KUKA KRL program: MyProgram_190().src

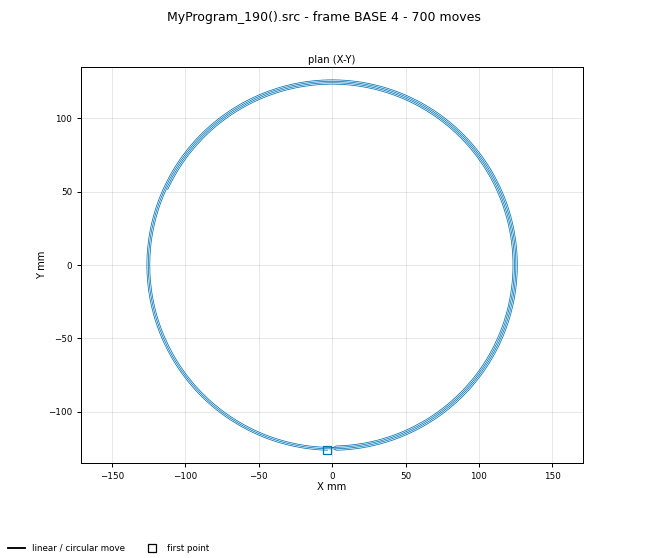
[picture p0: tool path of MyProgram_190().src in frame BASE 4, 700 of 700 moves have a stored position in this frame; points joined in program order, loops and branches not executed]
&ACCESS RVP
&REL 1
&PARAM TEMPLATE = C:\KRC\Roboter\Template\vorgabe
&PARAM EDITMASK = *
DEF MyProgram_190()
; ---- Setting reference (Base) ----
$BASE = BASE_DATA[4]

; --------------------------
; ---- Setting tool (TCP) ----
$TOOL = TOOL_DATA[3]
; --------------------------

$VEL.CP = VEL_APROX_PRINT
Startdeposition()
$VEL.CP = VEL_PRINT
LIN {X -3.1843,Y -126.111,Z 138,A -95.0934,B 24.9653,C -1.3617,E1 24.9951,E2 181.5075} C_DIS
LIN {X -7.0437,Y -125.9559,Z 138,A -96.9383,B 24.9655,C -1.3571,E1 24.9899,E2 183.3636} C_DIS
LIN {X -10.906,Y -125.6787,Z 138,A -98.6571,B 24.9654,C -1.3591,E1 24.9851,E2 185.0783} C_DIS
LIN {X -14.9041,Y -125.2671,Z 138,A -100.425,B 24.9652,C -1.3622,E1 24.9803,E2 186.8401} C_DIS
LIN {X -18.9665,Y -124.7171,Z 138,A -102.292,B 24.9652,C -1.3624,E1 24.9751,E2 188.7082} C_DIS
LIN {X -22.3988,Y -124.1462,Z 138,A -103.9323,B 24.9654,C -1.36,E1 24.9706,E2 190.3557} C_DIS
LIN {X -26.4694,Y -123.3424,Z 138,A -105.7239,B 24.9651,C -1.3653,E1 24.9657,E2 192.1369} C_DIS
LIN {X -29.6887,Y -122.6073,Z 138,A -107.3057,B 24.9652,C -1.3622,E1 24.9614,E2 193.7283} C_DIS
LIN {X -33.587,Y -121.5977,Z 138,A -108.947,B 24.9647,C -1.3723,E1 24.957,E2 195.3479} C_DIS
LIN {X -36.4143,Y -120.7816,Z 138,A -110.4707,B 24.9651,C -1.3643,E1 24.9529,E2 196.8933} C_DIS
LIN {X -39.9945,Y -119.6427,Z 138,A -112.121,B 24.9649,C -1.3683,E1 24.9485,E2 198.537} C_DIS
LIN {X -43.772,Y -118.3139,Z 138,A -113.9865,B 24.9649,C -1.3677,E1 24.9436,E2 200.4077} C_DIS
LIN {X -47.2767,Y -116.9565,Z 138,A -115.674,B 24.9649,C -1.3703,E1 24.9392,E2 202.0925} C_DIS
LIN {X -51.142,Y -115.3193,Z 138,A -117.5849,B 24.9647,C -1.3722,E1 24.9343,E2 204.0035} C_DIS
LIN {X -54.3155,Y -113.8583,Z 138,A -119.1216,B 24.9645,C -1.3765,E1 24.9304,E2 205.534} C_DIS
LIN {X -56.9474,Y -112.5654,Z 138,A -120.5382,B 24.9646,C -1.3741,E1 24.9269,E2 206.9598} C_DIS
LIN {X -61.2751,Y -110.2712,Z 138,A -122.6888,B 24.9643,C -1.3806,E1 24.9216,E2 209.1011} C_DIS
LIN {X -69.1084,Y -105.539,Z 138,A -127.0017,B 24.9643,C -1.3796,E1 24.9113,E2 213.4299} C_DIS
LIN {X -72.9275,Y -102.9369,Z 138,A -129.0758,B 24.9641,C -1.3843,E1 24.9066,E2 215.5} C_DIS
LIN {X -76.0268,Y -100.6691,Z 138,A -130.7644,B 24.9638,C -1.39,E1 24.9028,E2 217.181} C_DIS
LIN {X -78.4458,Y -98.7959,Z 138,A -132.3156,B 24.9641,C -1.385,E1 24.8994,E2 218.7496} C_DIS
LIN {X -82.0474,Y -95.8265,Z 138,A -134.3821,B 24.9637,C -1.3916,E1 24.8949,E2 220.8085} C_DIS
LIN {X -85.3051,Y -92.9376,Z 138,A -136.3149,B 24.9634,C -1.3977,E1 24.891,E2 222.7345} C_DIS
LIN {X -88.4698,Y -89.9305,Z 138,A -138.3203,B 24.9632,C -1.4009,E1 24.8869,E2 224.7408} C_DIS
LIN {X -91.4952,Y -86.8512,Z 138,A -140.3496,B 24.9632,C -1.402,E1 24.883,E2 226.776} C_DIS
LIN {X -94.065,Y -84.0604,Z 138,A -142.0826,B 24.963,C -1.4055,E1 24.8797,E2 228.5084} C_DIS
LIN {X -96.9286,Y -80.7424,Z 138,A -144.0584,B 24.9627,C -1.4109,E1 24.8762,E2 230.4805} C_DIS
LIN {X -99.5575,Y -77.4772,Z 138,A -145.9489,B 24.9624,C -1.4161,E1 24.8729,E2 232.3674} C_DIS
LIN {X -102.1418,Y -74.0365,Z 138,A -147.8756,B 24.9621,C -1.4223,E1 24.8697,E2 234.2887} C_DIS
LIN {X -104.5441,Y -70.6039,Z 138,A -149.8202,B 24.9619,C -1.4253,E1 24.8666,E2 236.2358} C_DIS
LIN {X -106.2939,Y -67.941,Z 138,A -151.3596,B 24.9619,C -1.4249,E1 24.8643,E2 237.7838} C_DIS
LIN {X -108.6351,Y -64.1314,Z 138,A -153.3025,B 24.9615,C -1.4344,E1 24.8615,E2 239.7142} C_DIS
LIN {X -110.5296,Y -60.8086,Z 138,A -155.0863,B 24.9613,C -1.4371,E1 24.8591,E2 241.5009} C_DIS
LIN {X -112.4396,Y -57.1946,Z 138,A -156.6495,B 24.9603,C -1.4556,E1 24.8571,E2 243.0282} C_DIS
LIN {X -114.1727,Y -53.6571,Z 138,A -158.7538,B 24.9608,C -1.4464,E1 24.8545,E2 245.1659} C_DIS
LIN {X -115.613,Y -50.4751,Z 138,A -160.2363,B 24.9603,C -1.4558,E1 24.8528,E2 246.6343} C_DIS
LIN {X -116.8237,Y -47.6062,Z 138,A -161.6588,B 24.9601,C -1.4595,E1 24.8513,E2 248.0557} C_DIS
LIN {X -118.3738,Y -43.612,Z 138,A -163.7518,B 24.9601,C -1.4587,E1 24.8492,E2 250.1624} C_DIS
LIN {X -119.6109,Y -40.0901,Z 138,A -165.3569,B 24.9596,C -1.468,E1 24.8478,E2 251.7547} C_DIS
LIN {X -120.5433,Y -37.193,Z 138,A -166.7446,B 24.9594,C -1.4719,E1 24.8466,E2 253.1408} C_DIS
LIN {X -121.4782,Y -34.0144,Z 138,A -168.2107,B 24.9591,C -1.4783,E1 24.8455,E2 254.6002} C_DIS
LIN {X -122.4907,Y -30.1723,Z 138,A -170.1494,B 24.9591,C -1.4779,E1 24.8441,E2 256.5511} C_DIS
LIN {X -123.8233,Y -24.1234,Z 138,A -172.9553,B 24.9586,C -1.4872,E1 24.8425,E2 259.3516} C_DIS
LIN {X -124.6687,Y -19.2791,Z 138,A -175.1858,B 24.9582,C -1.4945,E1 24.8415,E2 261.5779} C_DIS
LIN {X -125.1856,Y -15.5875,Z 138,A -176.8705,B 24.9578,C -1.5003,E1 24.8409,E2 263.2589} C_DIS
LIN {X -125.5705,Y -12.0845,Z 138,A -178.3017,B 24.9571,C -1.5131,E1 24.8405,E2 264.6681} C_DIS
LIN {X -125.7984,Y -9.4238,Z 138,A -179.776,B 24.9575,C -1.5053,E1 24.8401,E2 266.1698} C_DIS
LIN {X -126.0383,Y -5.3412,Z 138,A 178.3913,B 24.9571,C -1.5125,E1 24.8399,E2 267.9965} C_DIS
LIN {X -126.1439,Y -1.4652,Z 138,A 176.6709,B 24.9567,C -1.5201,E1 24.8398,E2 269.7091} C_DIS
LIN {X -126.1274,Y 2.4575,Z 138,A 174.9144,B 24.9563,C -1.527,E1 24.8398,E2 271.4596} C_DIS
LIN {X -125.9954,Y 6.2594,Z 138,A 173.1294,B 24.9561,C -1.5302,E1 24.84,E2 273.2478} C_DIS
LIN {X -125.7286,Y 10.3157,Z 138,A 171.4908,B 24.9552,C -1.5455,E1 24.8404,E2 274.8597} C_DIS
LIN {X -125.3625,Y 14.0922,Z 138,A 169.4724,B 24.9557,C -1.538,E1 24.8409,E2 276.9082} C_DIS
LIN {X -125.0413,Y 16.6956,Z 138,A 168.198,B 24.9557,C -1.5382,E1 24.8414,E2 278.1897} C_DIS
LIN {X -124.3839,Y 21.0404,Z 138,A 166.2733,B 24.9551,C -1.5479,E1 24.8423,E2 280.1028} C_DIS
LIN {X -123.728,Y 24.6098,Z 138,A 164.6559,B 24.9547,C -1.5546,E1 24.8431,E2 281.7136} C_DIS
LIN {X -123.0002,Y 28.0159,Z 138,A 162.8239,B 24.9551,C -1.5486,E1 24.8442,E2 283.5706} C_DIS
LIN {X -121.846,Y 32.6729,Z 138,A 160.8635,B 24.9541,C -1.5654,E1 24.8456,E2 285.5025} C_DIS
LIN {X -120.7193,Y 36.6178,Z 138,A 159.0027,B 24.9537,C -1.5715,E1 24.847,E2 287.3595} C_DIS
LIN {X -119.6782,Y 39.8879,Z 138,A 157.4553,B 24.9534,C -1.577,E1 24.8484,E2 288.9027} C_DIS
LIN {X -118.4195,Y 43.489,Z 138,A 155.6809,B 24.9532,C -1.5805,E1 24.85,E2 290.6787} C_DIS
LIN {X -117.115,Y 46.8834,Z 138,A 153.9246,B 24.9532,C -1.5811,E1 24.8518,E2 292.4437} C_DIS
LIN {X -115.3426,Y 51.0899,Z 138,A 152.1114,B 24.9521,C -1.5991,E1 24.8538,E2 294.2238} C_DIS
LIN {X -112.9708,Y 56.1391,Z 138,A 148.6942,B 24.954,C -1.5675,E1 24.8581,E2 297.735} C_DIS
LIN {X -110.5428,Y 60.7845,Z 138,A 146.6018,B 24.9528,C -1.5873,E1 24.8608,E2 299.7912} C_DIS
LIN {X -108.7408,Y 63.9515,Z 138,A 145.1814,B 24.9519,C -1.6026,E1 24.8628,E2 301.1824} C_DIS
LIN {X -106.4029,Y 67.7707,Z 138,A 143.1806,B 24.9514,C -1.61,E1 24.8657,E2 303.1759} C_DIS
LIN {X -103.8973,Y 71.5524,Z 138,A 141.1937,B 24.9509,C -1.6191,E1 24.8688,E2 305.1509} C_DIS
LIN {X -101.4707,Y 74.9543,Z 138,A 139.208,B 24.9508,C -1.6204,E1 24.8721,E2 307.1432} C_DIS
LIN {X -98.8671,Y 78.3563,Z 138,A 137.2836,B 24.9504,C -1.6267,E1 24.8754,E2 309.0618} C_DIS
LIN {X -96.2209,Y 81.5838,Z 138,A 135.3622,B 24.9502,C -1.6305,E1 24.8788,E2 310.9828} C_DIS
LIN {X -93.2585,Y 84.9545,Z 138,A 133.2981,B 24.9499,C -1.6346,E1 24.8826,E2 313.0465} C_DIS
LIN {X -90.3023,Y 88.0906,Z 138,A 131.3418,B 24.9496,C -1.6396,E1 24.8864,E2 314.9995} C_DIS
LIN {X -87.41,Y 90.9613,Z 138,A 129.4413,B 24.9495,C -1.6418,E1 24.8902,E2 316.9025} C_DIS
LIN {X -84.0588,Y 94.0664,Z 138,A 127.413,B 24.9491,C -1.6488,E1 24.8944,E2 318.9223} C_DIS
LIN {X -80.7619,Y 96.9125,Z 138,A 125.3839,B 24.9489,C -1.651,E1 24.8987,E2 320.9541} C_DIS
LIN {X -77.3811,Y 99.632,Z 138,A 123.4278,B 24.9486,C -1.656,E1 24.903,E2 322.9055} C_DIS
LIN {X -73.7304,Y 102.3636,Z 138,A 121.3155,B 24.9485,C -1.6585,E1 24.9077,E2 325.0194} C_DIS
LIN {X -70.0481,Y 104.9172,Z 138,A 119.304,B 24.9481,C -1.6636,E1 24.9124,E2 327.0253} C_DIS
LIN {X -66.2835,Y 107.3359,Z 138,A 117.2265,B 24.9481,C -1.6655,E1 24.9173,E2 329.1051} C_DIS
LIN {X -63.0471,Y 109.2678,Z 138,A 115.3202,B 24.9484,C -1.6597,E1 24.9219,E2 331.0309} C_DIS
LIN {X -60.2193,Y 110.8514,Z 138,A 114.0863,B 24.9475,C -1.6732,E1 24.9249,E2 332.2363} C_DIS
LIN {X -57.1335,Y 112.4707,Z 138,A 112.6236,B 24.947,C -1.6814,E1 24.9285,E2 333.6833} C_DIS
LIN {X -54.1653,Y 113.9301,Z 138,A 111.0462,B 24.947,C -1.6803,E1 24.9324,E2 335.2673} C_DIS
LIN {X -49.3542,Y 116.0976,Z 138,A 108.5307,B 24.9472,C -1.6784,E1 24.9389,E2 337.7935} C_DIS
LIN {X -45.9275,Y 117.4931,Z 138,A 106.9709,B 24.9467,C -1.6864,E1 24.9429,E2 339.3377} C_DIS
LIN {X -43.2268,Y 118.514,Z 138,A 105.6403,B 24.9467,C -1.6872,E1 24.9464,E2 340.669} C_DIS
LIN {X -37.0434,Y 120.5891,Z 138,A 102.7706,B 24.9462,C -1.6951,E1 24.954,E2 343.5252} C_DIS
LIN {X -34.1823,Y 121.4312,Z 138,A 101.3525,B 24.9462,C -1.6936,E1 24.9578,E2 344.9492} C_DIS
LIN {X -30.2186,Y 122.4795,Z 138,A 99.0393,B 24.9475,C -1.6744,E1 24.9642,E2 347.3115} C_DIS
LIN {X -26.6668,Y 123.2998,Z 138,A 97.5867,B 24.9468,C -1.6854,E1 24.9681,E2 348.7398} C_DIS
LIN {X -22.2034,Y 124.1812,Z 138,A 95.7017,B 24.9461,C -1.6955,E1 24.9732,E2 350.6026} C_DIS
LIN {X -18.2311,Y 124.8269,Z 138,A 93.8613,B 24.9461,C -1.6962,E1 24.9783,E2 352.4431} C_DIS
LIN {X -14.6843,Y 125.2933,Z 138,A 92.2052,B 24.9461,C -1.6957,E1 24.9829,E2 354.1015} C_DIS
LIN {X -10.7568,Y 125.6913,Z 138,A 90.446,B 24.946,C -1.6982,E1 24.9877,E2 355.8557} C_DIS
LIN {X -6.5893,Y 125.9788,Z 138,A 88.5503,B 24.946,C -1.699,E1 24.993,E2 357.7501} C_DIS
LIN {X -2.5849,Y 126.1252,Z 138,A 86.6906,B 24.946,C -1.6977,E1 24.9982,E2 359.6133} C_DIS
LIN {X 1.2278,Y 126.1459,Z 138,A 84.9358,B 24.946,C -1.6969,E1 25.0031,E2 361.3699} C_DIS
LIN {X 4.7952,Y 126.0596,Z 138,A 83.3843,B 24.9458,C -1.7004,E1 25.0074,E2 362.9127} C_DIS
LIN {X 8.6734,Y 125.8532,Z 138,A 81.5802,B 24.9459,C -1.6984,E1 25.0125,E2 364.7207} C_DIS
LIN {X 12.3307,Y 125.5469,Z 138,A 79.8631,B 24.9461,C -1.6958,E1 25.0173,E2 366.4429} C_DIS
LIN {X 16.3417,Y 125.0877,Z 138,A 78.1352,B 24.9458,C -1.7006,E1 25.022,E2 368.1583} C_DIS
LIN {X 20.3136,Y 124.5051,Z 138,A 76.2446,B 24.946,C -1.6967,E1 25.0273,E2 370.0561} C_DIS
LIN {X 23.9897,Y 123.8489,Z 138,A 74.5305,B 24.9461,C -1.6952,E1 25.032,E2 371.772} C_DIS
LIN {X 28.6252,Y 122.8611,Z 138,A 72.3822,B 24.9462,C -1.6943,E1 25.0378,E2 373.9197} C_DIS
LIN {X 32.2993,Y 121.9456,Z 138,A 70.8031,B 24.9458,C -1.7001,E1 25.0421,E2 375.4826} C_DIS
LIN {X 35.2724,Y 121.119,Z 138,A 69.395,B 24.9459,C -1.6987,E1 25.0458,E2 376.8914} C_DIS
LIN {X 38.3218,Y 120.1889,Z 138,A 67.8105,B 24.9464,C -1.6909,E1 25.0501,E2 378.4916} C_DIS
LIN {X 42.4475,Y 118.795,Z 138,A 65.9768,B 24.9461,C -1.6962,E1 25.0549,E2 380.3091} C_DIS
LIN {X 47.2661,Y 116.9608,Z 138,A 63.6076,B 24.9463,C -1.6925,E1 25.0611,E2 382.6818} C_DIS
LIN {X 50.697,Y 115.517,Z 138,A 61.8325,B 24.9467,C -1.6865,E1 25.0657,E2 384.4671} C_DIS
LIN {X 54.1241,Y 113.9497,Z 138,A 60.2039,B 24.9466,C -1.6885,E1 25.0698,E2 386.0866} C_DIS
LIN {X 59.137,Y 111.4316,Z 138,A 57.6397,B 24.9468,C -1.6843,E1 25.0761,E2 388.6537} C_DIS
LIN {X 61.5464,Y 110.1204,Z 138,A 55.6157,B 24.9493,C -1.6442,E1 25.0813,E2 390.7665} C_DIS
LIN {X 66.4381,Y 107.2399,Z 138,A 53.7538,B 24.9474,C -1.6755,E1 25.0855,E2 392.5486} C_DIS
LIN {X 70.3044,Y 104.7461,Z 138,A 51.6555,B 24.9476,C -1.6717,E1 25.0904,E2 394.6491} C_DIS
LIN {X 73.8549,Y 102.2734,Z 138,A 49.7166,B 24.9478,C -1.6696,E1 25.0948,E2 396.5862} C_DIS
LIN {X 77.3089,Y 99.6879,Z 138,A 47.8117,B 24.9478,C -1.6687,E1 25.0991,E2 398.4862} C_DIS
LIN {X 80.5283,Y 97.1059,Z 138,A 45.9147,B 24.9481,C -1.664,E1 25.1032,E2 400.3872} C_DIS
LIN {X 83.8428,Y 94.2597,Z 138,A 43.8929,B 24.9485,C -1.6581,E1 25.1074,E2 402.4149} C_DIS
LIN {X 86.381,Y 91.9388,Z 138,A 42.1429,B 24.9493,C -1.6454,E1 25.1111,E2 404.1877} C_DIS
LIN {X 88.7451,Y 89.6589,Z 138,A 40.8781,B 24.9488,C -1.6536,E1 25.1135,E2 405.4279} C_DIS
LIN {X 91.8682,Y 86.4558,Z 138,A 39.0098,B 24.9485,C -1.6573,E1 25.1171,E2 407.2793} C_DIS
LIN {X 94.718,Y 83.3243,Z 138,A 36.9318,B 24.9493,C -1.645,E1 25.121,E2 409.377} C_DIS
LIN {X 97.5231,Y 80.0228,Z 138,A 35.0003,B 24.9495,C -1.6421,E1 25.1245,E2 411.3065} C_DIS
LIN {X 100.1181,Y 76.7511,Z 138,A 33.2507,B 24.9493,C -1.6449,E1 25.1275,E2 413.0412} C_DIS
LIN {X 102.3611,Y 73.7339,Z 138,A 31.3767,B 24.9501,C -1.6321,E1 25.1306,E2 414.9364} C_DIS
LIN {X 104.915,Y 70.0514,Z 138,A 29.3991,B 24.9502,C -1.6298,E1 25.1337,E2 416.9097} C_DIS
LIN {X 107.3157,Y 66.3162,Z 138,A 27.3488,B 24.9507,C -1.6227,E1 25.1368,E2 418.9665} C_DIS
LIN {X 109.1543,Y 63.2431,Z 138,A 25.5345,B 24.9515,C -1.6087,E1 25.1394,E2 420.8045} C_DIS
LIN {X 110.7607,Y 60.3856,Z 138,A 24.3295,B 24.9509,C -1.619,E1 25.1409,E2 421.9788} C_DIS
LIN {X 114.4891,Y 52.973,Z 138,A 20.642,B 24.9513,C -1.6124,E1 25.1455,E2 425.6622} C_DIS
LIN {X 115.8897,Y 49.835,Z 138,A 19.048,B 24.9517,C -1.6061,E1 25.1473,E2 427.2622} C_DIS
LIN {X 117.448,Y 46.0433,Z 138,A 17.2365,B 24.9518,C -1.6032,E1 25.1492,E2 429.0707} C_DIS
LIN {X 118.7956,Y 42.4458,Z 138,A 15.2611,B 24.9529,C -1.5861,E1 25.1511,E2 431.0754} C_DIS
LIN {X 120.1635,Y 38.4011,Z 138,A 13.4636,B 24.9528,C -1.5874,E1 25.1526,E2 432.8595} C_DIS
LIN {X 121.6807,Y 33.2905,Z 138,A 11.0418,B 24.9532,C -1.5799,E1 25.1545,E2 435.2853} C_DIS
LIN {X 122.6042,Y 29.7014,Z 138,A 9.4799,B 24.9532,C -1.5809,E1 25.1556,E2 436.8358} C_DIS
LIN {X 123.5258,Y 25.6034,Z 138,A 7.5395,B 24.9536,C -1.5731,E1 25.1567,E2 438.7832} C_DIS
LIN {X 124.1856,Y 22.179,Z 138,A 6.0159,B 24.9537,C -1.5712,E1 25.1575,E2 440.3024} C_DIS
LIN {X 124.8109,Y 18.3432,Z 138,A 4.1928,B 24.9543,C -1.5625,E1 25.1583,E2 442.1353} C_DIS
LIN {X 125.3007,Y 14.6229,Z 138,A 2.492,B 24.9546,C -1.5572,E1 25.1589,E2 443.8386} C_DIS
LIN {X 125.7021,Y 10.6293,Z 138,A 0.7505,B 24.9546,C -1.5555,E1 25.1593,E2 445.5738} C_DIS
LIN {X 125.9762,Y 6.6414,Z 138,A -1.0667,B 24.955,C -1.5494,E1 25.1596,E2 447.3944} C_DIS
LIN {X 126.1201,Y 2.8566,Z 138,A -2.8293,B 24.9555,C -1.5416,E1 25.1598,E2 449.165} C_DIS
LIN {X 126.1503,Y -0.69,Z 138,A -4.4682,B 24.9559,C -1.5348,E1 25.1598,E2 450.8101} C_DIS
LIN {X 126.0556,Y -4.899,Z 138,A -6.2874,B 24.9559,C -1.5334,E1 25.1596,E2 452.6219} C_DIS
LIN {X 125.8258,Y -9.049,Z 138,A -8.1294,B 24.9562,C -1.5295,E1 25.1593,E2 454.462} C_DIS
LIN {X 125.4968,Y -12.8441,Z 138,A -9.9084,B 24.9566,C -1.5213,E1 25.1588,E2 456.2499} C_DIS
LIN {X 125.0537,Y -16.6009,Z 138,A -11.5281,B 24.9566,C -1.5208,E1 25.1583,E2 457.8613} C_DIS
LIN {X 124.4813,Y -20.4567,Z 138,A -13.2807,B 24.957,C -1.5159,E1 25.1575,E2 459.6152} C_DIS
LIN {X 123.8791,Y -23.8316,Z 138,A -14.866,B 24.9573,C -1.5093,E1 25.1567,E2 461.2066} C_DIS
LIN {X 123.2436,Y -26.9272,Z 138,A -16.5653,B 24.9584,C -1.4909,E1 25.1557,E2 462.9394} C_DIS
LIN {X 121.9819,Y -32.1631,Z 138,A -18.7377,B 24.958,C -1.4972,E1 25.1542,E2 465.0844} C_DIS
LIN {X 121.0599,Y -35.4744,Z 138,A -20.6849,B 24.9594,C -1.4722,E1 25.1527,E2 467.0795} C_DIS
LIN {X 119.8982,Y -39.2273,Z 138,A -21.9524,B 24.9582,C -1.4932,E1 25.1517,E2 468.2903} C_DIS
LIN {X 118.1968,Y -44.0845,Z 138,A -24.2966,B 24.9587,C -1.4854,E1 25.1495,E2 470.6396} C_DIS
LIN {X 117.0448,Y -47.0577,Z 138,A -25.8717,B 24.9593,C -1.4743,E1 25.1478,E2 472.2323} C_DIS
LIN {X 115.4048,Y -50.9508,Z 138,A -27.6176,B 24.9591,C -1.4773,E1 25.1459,E2 473.9616} C_DIS
LIN {X 114.032,Y -53.9519,Z 138,A -29.2873,B 24.9599,C -1.4638,E1 25.1439,E2 475.6539} C_DIS
LIN {X 112.424,Y -57.2252,Z 138,A -30.8725,B 24.9599,C -1.4624,E1 25.142,E2 477.2339} C_DIS
LIN {X 110.6036,Y -60.6736,Z 138,A -32.6818,B 24.9603,C -1.4551,E1 25.1395,E2 479.051} C_DIS
LIN {X 108.4198,Y -64.4944,Z 138,A -34.6472,B 24.9606,C -1.4509,E1 25.1368,E2 481.0161} C_DIS
LIN {X 106.0835,Y -68.2696,Z 138,A -36.6913,B 24.961,C -1.4436,E1 25.1337,E2 483.0671} C_DIS
LIN {X 103.7128,Y -71.8198,Z 138,A -38.6197,B 24.9612,C -1.4387,E1 25.1307,E2 484.9977} C_DIS
LIN {X 101.248,Y -75.2542,Z 138,A -41.247,B 24.9634,C -1.3971,E1 25.1262,E2 487.7104} C_DIS
LIN {X 97.6826,Y -79.8276,Z 138,A -42.915,B 24.9612,C -1.4394,E1 25.1235,E2 489.2707} C_DIS
LIN {X 93.6621,Y -84.5097,Z 138,A -45.9515,B 24.9622,C -1.42,E1 25.1178,E2 492.3394} C_DIS
LIN {X 90.972,Y -87.3988,Z 138,A -47.6004,B 24.9621,C -1.4228,E1 25.1147,E2 493.9745} C_DIS
LIN {X 88.0571,Y -90.335,Z 138,A -49.9829,B 24.9637,C -1.3924,E1 25.1098,E2 496.4186} C_DIS
LIN {X 85.0001,Y -93.2171,Z 138,A -51.4919,B 24.9629,C -1.4082,E1 25.1068,E2 497.8843} C_DIS
LIN {X 81.6866,Y -96.1335,Z 138,A -53.4312,B 24.9629,C -1.4069,E1 25.1027,E2 499.8191} C_DIS
LIN {X 79.4361,Y -98.0018,Z 138,A -55.2722,B 24.9644,C -1.3778,E1 25.0986,E2 501.7217} C_DIS
LIN {X 75.8471,Y -100.8048,Z 138,A -56.7504,B 24.9631,C -1.4033,E1 25.0955,E2 503.1345} C_DIS
LIN {X 73.2379,Y -102.716,Z 138,A -58.6682,B 24.9645,C -1.3774,E1 25.091,E2 505.1067} C_DIS
LIN {X 69.9914,Y -104.955,Z 138,A -60.4202,B 24.9645,C -1.3758,E1 25.0869,E2 506.8567} C_DIS
LIN {X 66.7977,Y -107.0161,Z 138,A -61.7787,B 24.9638,C -1.391,E1 25.0838,E2 508.1748} C_DIS
LIN {X 63.2431,Y -109.1543,Z 138,A -63.7237,B 24.9641,C -1.3844,E1 25.0791,E2 510.1295} C_DIS
LIN {X 59.2938,Y -111.3493,Z 138,A -65.803,B 24.9644,C -1.3794,E1 25.074,E2 512.2146} C_DIS
LIN {X 56.0006,Y -113.0392,Z 138,A -67.2995,B 24.964,C -1.3859,E1 25.0703,E2 513.6917} C_DIS
LIN {X 53.0828,Y -114.4383,Z 138,A -68.672,B 24.9639,C -1.3884,E1 25.0669,E2 515.0547} C_DIS
LIN {X 50.3542,Y -115.6652,Z 138,A -70.1541,B 24.9643,C -1.3801,E1 25.063,E2 516.5528} C_DIS
LIN {X 47.3312,Y -116.9345,Z 138,A -71.6241,B 24.9643,C -1.3789,E1 25.0593,E2 518.0223} C_DIS
LIN {X 41.9125,Y -118.9859,Z 138,A -74.2561,B 24.9646,C -1.3753,E1 25.0524,E2 520.6574} C_DIS
LIN {X 38.2727,Y -120.2045,Z 138,A -75.9935,B 24.9646,C -1.3734,E1 25.0477,E2 522.3958} C_DIS
LIN {X 32.7287,Y -121.8311,Z 138,A -78.6274,B 24.9648,C -1.37,E1 25.0407,E2 525.0334} C_DIS
LIN {X 28.7378,Y -122.8353,Z 138,A -80.5606,B 24.9651,C -1.3649,E1 25.0354,E2 526.9759} C_DIS
LIN {X 25.136,Y -123.6209,Z 138,A -82.2903,B 24.9653,C -1.3606,E1 25.0306,E2 528.7134} C_DIS
LIN {X 20.8141,Y -124.4216,Z 138,A -84.0653,B 24.9648,C -1.37,E1 25.0258,E2 530.4644} C_DIS
LIN {X 17.6706,Y -124.907,Z 138,A -85.5773,B 24.9651,C -1.3656,E1 25.0216,E2 531.9853} C_DIS
LIN {X 13.8266,Y -125.3911,Z 138,A -87.3421,B 24.9651,C -1.3643,E1 25.0167,E2 533.7519} C_DIS
LIN {X 10.3306,Y -125.7273,Z 138,A -89.0133,B 24.9654,C -1.3597,E1 25.0121,E2 535.433} C_DIS
LIN {X 6.5028,Y -125.9831,Z 138,A -90.6761,B 24.9652,C -1.3629,E1 25.0074,E2 537.0877} C_DIS
LIN {X 2.7912,Y -126.1218,Z 138,A -92.4593,B 24.9655,C -1.3576,E1 25.0024,E2 538.883} C_DIS
LIN {X 2.7912,Y -126.1218,Z 138,A -92.4593,B 24.9655,C -1.3576,E1 25.0024,E2 538.883} C_DIS
Enddeposition()
LIN {X 0.8852,Y -125.1643,Z 138,A -93.1588,B 24.9642,C -1.3828,E1 25.0007,E2 539.5227} C_DIS
Startdeposition()
$VEL.CP = VEL_PRINT
LIN {X 3.3988,Y -125.1228,Z 138,A -91.394,B 24.9626,C -1.4132,E1 25.0058,E2 537.6863} C_DIS
LIN {X 7.3779,Y -124.9516,Z 138,A -89.5453,B 24.9625,C -1.4152,E1 25.0109,E2 535.8334} C_DIS
LIN {X 11.1676,Y -124.6712,Z 138,A -87.7011,B 24.9622,C -1.4212,E1 25.0161,E2 533.9759} C_DIS
LIN {X 15.0926,Y -124.2558,Z 138,A -85.9375,B 24.9622,C -1.4202,E1 25.021,E2 532.2161} C_DIS
LIN {X 19.2045,Y -123.6867,Z 138,A -84.1263,B 24.9624,C -1.4171,E1 25.026,E2 530.4137} C_DIS
LIN {X 23.2174,Y -122.9969,Z 138,A -82.0486,B 24.9617,C -1.4293,E1 25.0317,E2 528.3095} C_DIS
LIN {X 27.4372,Y -122.1253,Z 138,A -80.4647,B 24.9627,C -1.4117,E1 25.036,E2 526.7693} C_DIS
LIN {X 30.6364,Y -121.3615,Z 138,A -78.8102,B 24.9622,C -1.4206,E1 25.0405,E2 525.096} C_DIS
LIN {X 38.0234,Y -119.2534,Z 138,A -75.3255,B 24.9621,C -1.423,E1 25.0498,E2 521.6117} C_DIS
LIN {X 44.3504,Y -117.0488,Z 138,A -72.261,B 24.9619,C -1.4269,E1 25.0579,E2 518.5443} C_DIS
LIN {X 48.0056,Y -115.597,Z 138,A -70.3888,B 24.9615,C -1.4331,E1 25.0628,E2 516.6616} C_DIS
LIN {X 51.5068,Y -114.0805,Z 138,A -68.7642,B 24.9617,C -1.4296,E1 25.0669,E2 515.0492} C_DIS
LIN {X 54.1038,Y -112.8713,Z 138,A -67.398,B 24.9614,C -1.4345,E1 25.0704,E2 513.6749} C_DIS
LIN {X 57.3557,Y -111.2558,Z 138,A -65.6064,B 24.9609,C -1.4439,E1 25.0749,E2 511.8661} C_DIS
LIN {X 63.1409,Y -108.0782,Z 138,A -62.6695,B 24.9609,C -1.4451,E1 25.082,E2 508.9352} C_DIS
LIN {X 66.5896,Y -105.9881,Z 138,A -60.8077,B 24.9606,C -1.4494,E1 25.0864,E2 507.069} C_DIS
LIN {X 69.6045,Y -104.0327,Z 138,A -58.7802,B 24.9594,C -1.4724,E1 25.0913,E2 504.994} C_DIS
LIN {X 72.9163,Y -101.739,Z 138,A -57.6001,B 24.961,C -1.4421,E1 25.0938,E2 503.8894} C_DIS
LIN {X 75.1,Y -100.1385,Z 138,A -56.0972,B 24.9602,C -1.4583,E1 25.0972,E2 502.3537} C_DIS
LIN {X 79.9228,Y -96.3325,Z 138,A -52.699,B 24.9581,C -1.4949,E1 25.1047,E2 498.882} C_DIS
LIN {X 83.7699,Y -93.0071,Z 138,A -51.1055,B 24.9599,C -1.4624,E1 25.1079,E2 497.3716} C_DIS
LIN {X 88.404,Y -88.6137,Z 138,A -48.3499,B 24.96,C -1.4608,E1 25.1134,E2 494.631} C_DIS
LIN {X 92.6399,Y -84.1751,Z 138,A -45.3753,B 24.9592,C -1.4765,E1 25.1192,E2 491.6324} C_DIS
LIN {X 96.577,Y -79.6275,Z 138,A -42.6928,B 24.959,C -1.4801,E1 25.124,E2 488.9537} C_DIS
LIN {X 100.1693,Y -75.059,Z 138,A -40.1585,B 24.959,C -1.4808,E1 25.1284,E2 486.4296} C_DIS
LIN {X 101.7027,Y -72.967,Z 138,A -38.7235,B 24.958,C -1.497,E1 25.1308,E2 484.9635} C_DIS
LIN {X 104.0523,Y -69.5752,Z 138,A -36.8343,B 24.9577,C -1.5024,E1 25.1337,E2 483.0708} C_DIS
LIN {X 106.3973,Y -65.9337,Z 138,A -34.8597,B 24.9574,C -1.5077,E1 25.1367,E2 481.0937} C_DIS
LIN {X 108.4615,Y -62.48,Z 138,A -33.0225,B 24.9571,C -1.5129,E1 25.1393,E2 479.2536} C_DIS
LIN {X 110.1462,Y -59.4599,Z 138,A -31.4785,B 24.957,C -1.5156,E1 25.1413,E2 477.7113} C_DIS
LIN {X 112.0758,Y -55.7342,Z 138,A -29.6105,B 24.9568,C -1.5187,E1 25.1437,E2 475.8459} C_DIS
LIN {X 113.6426,Y -52.4642,Z 138,A -27.9747,B 24.9566,C -1.5226,E1 25.1456,E2 474.2099} C_DIS
LIN {X 115.874,Y -47.3359,Z 138,A -25.5598,B 24.9566,C -1.5229,E1 25.1483,E2 471.8074} C_DIS
LIN {X 117.391,Y -43.4367,Z 138,A -23.4333,B 24.9556,C -1.54,E1 25.1504,E2 469.6524} C_DIS
LIN {X 118.9827,Y -38.8687,Z 138,A -20.8684,B 24.9541,C -1.5655,E1 25.1527,E2 467.042} C_DIS
LIN {X 120.1431,Y -35.1112,Z 138,A -19.5632,B 24.9553,C -1.5453,E1 25.1537,E2 465.7918} C_DIS
LIN {X 121.1599,Y -31.4309,Z 138,A -16.993,B 24.9524,C -1.5942,E1 25.1556,E2 463.1212} C_DIS
LIN {X 122.4816,Y -25.8039,Z 138,A -15.2459,B 24.9547,C -1.5555,E1 25.1566,E2 461.4755} C_DIS
LIN {X 123.069,Y -22.84,Z 138,A -13.7051,B 24.9539,C -1.5683,E1 25.1574,E2 459.9136} C_DIS
LIN {X 123.6896,Y -19.1858,Z 138,A -12.1303,B 24.9539,C -1.5675,E1 25.1581,E2 458.3499} C_DIS
LIN {X 124.2349,Y -15.2682,Z 138,A -10.2593,B 24.9534,C -1.5766,E1 25.1588,E2 456.4684} C_DIS
LIN {X 124.6082,Y -11.8335,Z 138,A -8.7572,B 24.9534,C -1.5777,E1 25.1592,E2 454.9727} C_DIS
LIN {X 124.9277,Y -7.7667,Z 138,A -6.9056,B 24.953,C -1.583,E1 25.1595,E2 453.1195} C_DIS
LIN {X 125.1138,Y -3.7217,Z 138,A -5.0474,B 24.9527,C -1.5893,E1 25.1597,E2 451.2574} C_DIS
LIN {X 125.1709,Y 0.3093,Z 138,A -3.1114,B 24.952,C -1.6001,E1 25.1597,E2 449.3075} C_DIS
LIN {X 125.0876,Y 4.5231,Z 138,A -1.285,B 24.952,C -1.6011,E1 25.1597,E2 447.4897} C_DIS
LIN {X 124.9014,Y 8.1939,Z 138,A 0.4591,B 24.9514,C -1.6098,E1 25.1593,E2 445.7354} C_DIS
LIN {X 124.5576,Y 12.3608,Z 138,A 2.3148,B 24.9512,C -1.613,E1 25.1589,E2 443.8832} C_DIS
LIN {X 124.0998,Y 16.3235,Z 138,A 4.0783,B 24.9511,C -1.6157,E1 25.1583,E2 442.1238} C_DIS
LIN {X 123.5001,Y 20.3713,Z 138,A 5.9435,B 24.9507,C -1.6213,E1 25.1575,E2 440.2563} C_DIS
LIN {X 122.8681,Y 23.8913,Z 138,A 7.5185,B 24.9507,C -1.6233,E1 25.1567,E2 438.6858} C_DIS
LIN {X 121.618,Y 29.6027,Z 138,A 10.2485,B 24.9499,C -1.6345,E1 25.155,E2 435.9452} C_DIS
LIN {X 120.4956,Y 33.8823,Z 138,A 12.2251,B 24.9497,C -1.6383,E1 25.1535,E2 433.9711} C_DIS
LIN {X 119.0789,Y 38.5698,Z 138,A 14.727,B 24.9484,C -1.6587,E1 25.1514,E2 431.4352} C_DIS
LIN {X 117.7186,Y 42.5381,Z 138,A 16.3451,B 24.9491,C -1.6488,E1 25.1499,E2 429.8495} C_DIS
LIN {X 116.6383,Y 45.4165,Z 138,A 17.7306,B 24.9489,C -1.6519,E1 25.1486,E2 428.4644} C_DIS
LIN {X 115.4103,Y 48.4525,Z 138,A 19.2404,B 24.9486,C -1.6569,E1 25.1469,E2 426.9512} C_DIS
LIN {X 113.7665,Y 52.1963,Z 138,A 21.5547,B 24.9468,C -1.6853,E1 25.1442,E2 424.5825} C_DIS
LIN {X 112.0869,Y 55.7105,Z 138,A 23.1258,B 24.9471,C -1.6794,E1 25.1423,E2 423.0337} C_DIS
LIN {X 109.8628,Y 59.9812,Z 138,A 25.1711,B 24.9473,C -1.6773,E1 25.1396,E2 421.0041} C_DIS
LIN {X 108.0782,Y 63.1409,Z 138,A 26.6583,B 24.9476,C -1.6729,E1 25.1376,E2 419.5349} C_DIS
LIN {X 106.2185,Y 66.221,Z 138,A 28.4048,B 24.947,C -1.6825,E1 25.135,E2 417.7747} C_DIS
LIN {X 103.8755,Y 69.8399,Z 138,A 30.2827,B 24.947,C -1.6828,E1 25.1321,E2 415.9056} C_DIS
LIN {X 101.78,Y 72.8589,Z 138,A 32.1503,B 24.9461,C -1.6966,E1 25.1291,E2 414.0145} C_DIS
LIN {X 99.4066,Y 76.0652,Z 138,A 33.8698,B 24.9461,C -1.6957,E1 25.1262,E2 412.3053} C_DIS
LIN {X 96.6734,Y 79.5109,Z 138,A 35.9215,B 24.9457,C -1.7025,E1 25.1226,E2 410.247} C_DIS
LIN {X 93.8905,Y 82.778,Z 138,A 37.8845,B 24.9454,C -1.7071,E1 25.119,E2 408.2821} C_DIS
LIN {X 91.4117,Y 85.5076,Z 138,A 39.5364,B 24.9453,C -1.7091,E1 25.1159,E2 406.6327} C_DIS
LIN {X 88.4388,Y 88.5791,Z 138,A 41.5082,B 24.9449,C -1.7142,E1 25.112,E2 404.6573} C_DIS
LIN {X 85.5998,Y 91.3259,Z 138,A 43.1344,B 24.9453,C -1.7088,E1 25.1088,E2 403.0507} C_DIS
LIN {X 83.0878,Y 93.6166,Z 138,A 44.8335,B 24.9446,C -1.7192,E1 25.1052,E2 401.3338} C_DIS
LIN {X 80.288,Y 96.0285,Z 138,A 46.5062,B 24.9445,C -1.7216,E1 25.1016,E2 399.662} C_DIS
LIN {X 76.9773,Y 98.7027,Z 138,A 48.4957,B 24.9441,C -1.7273,E1 25.0973,E2 397.6663} C_DIS
LIN {X 73.5201,Y 101.3035,Z 138,A 50.399,B 24.9441,C -1.727,E1 25.093,E2 395.7706} C_DIS
LIN {X 70.0082,Y 103.7616,Z 138,A 52.4523,B 24.9436,C -1.7349,E1 25.0882,E2 393.7055} C_DIS
LIN {X 67.1383,Y 105.6418,Z 138,A 53.9634,B 24.9436,C -1.7344,E1 25.0847,E2 392.2005} C_DIS
LIN {X 61.814,Y 108.8425,Z 138,A 56.9098,B 24.943,C -1.7438,E1 25.0776,E2 389.2409} C_DIS
LIN {X 57.8001,Y 111.0246,Z 138,A 58.7916,B 24.9435,C -1.7362,E1 25.073,E2 387.3824} C_DIS
LIN {X 54.442,Y 112.7097,Z 138,A 60.3649,B 24.9438,C -1.7311,E1 25.0691,E2 385.8252} C_DIS
LIN {X 50.9928,Y 114.3104,Z 138,A 62.2168,B 24.9433,C -1.7387,E1 25.0644,E2 383.9601} C_DIS
LIN {X 47.788,Y 115.6879,Z 138,A 63.9008,B 24.9429,C -1.7448,E1 25.06,E2 382.2657} C_DIS
LIN {X 43.7778,Y 117.2632,Z 138,A 65.7668,B 24.9432,C -1.7415,E1 25.0552,E2 380.4116} C_DIS
LIN {X 40.6057,Y 118.3998,Z 138,A 67.446,B 24.9426,C -1.7496,E1 25.0507,E2 378.7165} C_DIS
LIN {X 36.0806,Y 119.8569,Z 138,A 69.473,B 24.943,C -1.744,E1 25.0453,E2 376.7065} C_DIS
LIN {X 32.4553,Y 120.8878,Z 138,A 71.2501,B 24.9428,C -1.7477,E1 25.0405,E2 374.9235} C_DIS
LIN {X 28.8802,Y 121.7922,Z 138,A 73.3085,B 24.9415,C -1.7668,E1 25.0348,E2 372.8227} C_DIS
LIN {X 25.3435,Y 122.5767,Z 138,A 74.5545,B 24.9428,C -1.7475,E1 25.0316,E2 371.6242} C_DIS
LIN {X 21.7261,Y 123.2691,Z 138,A 76.3001,B 24.9425,C -1.751,E1 25.0268,E2 369.8721} C_DIS
LIN {X 17.7917,Y 123.8978,Z 138,A 78.0709,B 24.9427,C -1.749,E1 25.0219,E2 368.1077} C_DIS
LIN {X 14.0881,Y 124.3754,Z 138,A 79.8997,B 24.9423,C -1.7551,E1 25.0168,E2 366.2659} C_DIS
LIN {X 10.2251,Y 124.7509,Z 138,A 81.6722,B 24.9423,C -1.7551,E1 25.0118,E2 364.4944} C_DIS
LIN {X 6.1929,Y 125.0156,Z 138,A 83.4612,B 24.9425,C -1.7522,E1 25.0069,E2 362.7131} C_DIS
LIN {X 2.0825,Y 125.1516,Z 138,A 85.3138,B 24.9425,C -1.7505,E1 25.0017,E2 360.8647} C_DIS
LIN {X -1.8898,Y 125.1548,Z 138,A 87.1218,B 24.9426,C -1.7496,E1 24.9967,E2 359.0588} C_DIS
LIN {X -5.6031,Y 125.0453,Z 138,A 88.9332,B 24.9423,C -1.7544,E1 24.9916,E2 357.2358} C_DIS
LIN {X -9.4431,Y 124.8126,Z 138,A 90.6846,B 24.9423,C -1.7532,E1 24.9867,E2 355.4866} C_DIS
LIN {X -13.5441,Y 124.4339,Z 138,A 92.4011,B 24.943,C -1.7442,E1 24.982,E2 353.7905} C_DIS
LIN {X -16.884,Y 124.0263,Z 138,A 94.0154,B 24.9428,C -1.7467,E1 24.9775,E2 352.169} C_DIS
LIN {X -20.5832,Y 123.4647,Z 138,A 95.6838,B 24.943,C -1.7434,E1 24.9729,E2 350.5069} C_DIS
LIN {X -23.745,Y 122.896,Z 138,A 97.9021,B 24.9408,C -1.7778,E1 24.9666,E2 348.2045} C_DIS
LIN {X -28.8103,Y 121.809,Z 138,A 99.6942,B 24.9427,C -1.748,E1 24.9619,E2 346.4808} C_DIS
LIN {X -33.3212,Y 120.6525,Z 138,A 101.7087,B 24.9432,C -1.7403,E1 24.9565,E2 344.4816} C_DIS
LIN {X -37.4264,Y 119.4433,Z 138,A 104.278,B 24.9415,C -1.7668,E1 24.9495,E2 341.8449} C_DIS
LIN {X -41.8571,Y 117.9641,Z 138,A 105.7262,B 24.9438,C -1.7316,E1 24.9459,E2 340.4774} C_DIS
LIN {X -45.5277,Y 116.5951,Z 138,A 107.6164,B 24.9437,C -1.7338,E1 24.9409,E2 338.5782} C_DIS
LIN {X -48.3677,Y 115.4458,Z 138,A 108.9651,B 24.944,C -1.7293,E1 24.9375,E2 337.2372} C_DIS
LIN {X -52.9662,Y 113.4105,Z 138,A 111.6737,B 24.943,C -1.7447,E1 24.9305,E2 334.4853} C_DIS
LIN {X -56.0939,Y 111.8981,Z 138,A 112.8956,B 24.9442,C -1.7249,E1 24.9275,E2 333.3072} C_DIS
LIN {X -58.4282,Y 110.6947,Z 138,A 115.0053,B 24.9416,C -1.7652,E1 24.9221,E2 331.0957} C_DIS
LIN {X -63.6849,Y 107.7587,Z 138,A 116.6992,B 24.9452,C -1.7107,E1 24.9183,E2 329.5265} C_DIS
LIN {X -67.8275,Y 105.2006,Z 138,A 119.2703,B 24.9444,C -1.7223,E1 24.9121,E2 326.9197} C_DIS
LIN {X -71.5466,Y 102.7068,Z 138,A 121.258,B 24.9449,C -1.7153,E1 24.9076,E2 324.942} C_DIS
LIN {X -74.626,Y 100.4916,Z 138,A 122.9961,B 24.9451,C -1.7117,E1 24.9036,E2 323.2062} C_DIS
LIN {X -77.7674,Y 98.0809,Z 138,A 124.8688,B 24.9451,C -1.7105,E1 24.8995,E2 321.3294} C_DIS
LIN {X -81.3125,Y 95.1628,Z 138,A 126.9493,B 24.9455,C -1.7048,E1 24.8951,E2 319.2547} C_DIS
LIN {X -84.4636,Y 92.3774,Z 138,A 128.9338,B 24.9456,C -1.703,E1 24.891,E2 317.2664} C_DIS
LIN {X -87.74,Y 89.2709,Z 138,A 130.9652,B 24.9461,C -1.6964,E1 24.8869,E2 315.2423} C_DIS
LIN {X -90.7879,Y 86.1701,Z 138,A 133.0184,B 24.9462,C -1.6943,E1 24.8829,E2 313.1853} C_DIS
LIN {X -93.8024,Y 82.8776,Z 138,A 135.0347,B 24.9466,C -1.6878,E1 24.8791,E2 311.1755} C_DIS
LIN {X -96.681,Y 79.5017,Z 138,A 137.0972,B 24.9469,C -1.6839,E1 24.8754,E2 309.1129} C_DIS
LIN {X -99.329,Y 76.1667,Z 138,A 139.0421,B 24.9472,C -1.6784,E1 24.8721,E2 307.1717} C_DIS
LIN {X -102.0454,Y 72.4878,Z 138,A 141.0923,B 24.9477,C -1.6706,E1 24.8688,E2 305.1302} C_DIS
LIN {X -104.3532,Y 69.1239,Z 138,A 143.0431,B 24.9477,C -1.6691,E1 24.8657,E2 303.1732} C_DIS
LIN {X -106.5487,Y 65.689,Z 138,A 145.2948,B 24.947,C -1.6812,E1 24.8623,E2 300.8811} C_DIS
LIN {X -108.6143,Y 62.2134,Z 138,A 146.6833,B 24.9487,C -1.6548,E1 24.8605,E2 299.5484} C_DIS
LIN {X -110.7423,Y 58.3377,Z 138,A 148.7973,B 24.9488,C -1.6529,E1 24.8577,E2 297.4278} C_DIS
LIN {X -112.4232,Y 55.0299,Z 138,A 150.523,B 24.949,C -1.6489,E1 24.8555,E2 295.7021} C_DIS
LIN {X -114.3874,Y 50.8207,Z 138,A 152.569,B 24.9497,C -1.6388,E1 24.8532,E2 293.6691} C_DIS
LIN {X -116.4821,Y 45.8183,Z 138,A 154.9102,B 24.9505,C -1.6247,E1 24.8507,E2 291.3485} C_DIS
LIN {X -117.794,Y 42.3289,Z 138,A 156.8078,B 24.9503,C -1.6279,E1 24.8488,E2 289.4325} C_DIS
LIN {X -119.1426,Y 38.3703,Z 138,A 158.7197,B 24.9507,C -1.6217,E1 24.8472,E2 287.5244} C_DIS
LIN {X -120.2163,Y 34.8614,Z 138,A 160.4996,B 24.9507,C -1.6209,E1 24.8457,E2 285.7364} C_DIS
LIN {X -121.299,Y 30.8827,Z 138,A 162.2574,B 24.9515,C -1.6089,E1 24.8445,E2 283.9967} C_DIS
LIN {X -122.77,Y 24.3937,Z 138,A 165.2405,B 24.9523,C -1.5962,E1 24.8427,E2 281.0266} C_DIS
LIN {X -123.5196,Y 20.2542,Z 138,A 167.8946,B 24.9507,C -1.6227,E1 24.8415,E2 278.2933} C_DIS
LIN {X -124.1862,Y 15.6644,Z 138,A 169.4334,B 24.9527,C -1.5893,E1 24.8409,E2 276.825} C_DIS
LIN {X -124.7832,Y 9.8421,Z 138,A 172.1126,B 24.9532,C -1.5805,E1 24.8402,E2 274.1507} C_DIS
LIN {X -125.0082,Y 6.3393,Z 138,A 173.7709,B 24.9534,C -1.5776,E1 24.8399,E2 272.4894} C_DIS
LIN {X -125.1681,Y 0.734,Z 138,A 176.606,B 24.9532,C -1.5812,E1 24.8398,E2 269.6286} C_DIS
LIN {X -125.1233,Y -3.379,Z 138,A 178.2362,B 24.9542,C -1.5637,E1 24.8398,E2 268.0304} C_DIS
LIN {X -124.9913,Y -6.676,Z 138,A -179.9656,B 24.9537,C -1.5717,E1 24.8401,E2 266.2022} C_DIS
LIN {X -124.451,Y -13.3857,Z 138,A -177.1679,B 24.9551,C -1.5489,E1 24.8408,E2 263.4421} C_DIS
LIN {X -124.0767,Y -16.5001,Z 138,A -175.6995,B 24.9552,C -1.5457,E1 24.8413,E2 261.9725} C_DIS
LIN {X -123.0019,Y -23.191,Z 138,A -172.6519,B 24.956,C -1.5333,E1 24.8428,E2 258.9365} C_DIS
LIN {X -121.7759,Y -28.9477,Z 138,A -169.9955,B 24.9565,C -1.523,E1 24.8443,E2 256.2889} C_DIS
LIN {X -120.867,Y -32.5333,Z 138,A -168.2098,B 24.9566,C -1.5219,E1 24.8456,E2 254.4955} C_DIS
LIN {X -120.0558,Y -35.4093,Z 138,A -166.7623,B 24.9566,C -1.5213,E1 24.8467,E2 253.041} C_DIS
LIN {X -118.8394,Y -39.2992,Z 138,A -164.8501,B 24.9568,C -1.5177,E1 24.8483,E2 251.1264} C_DIS
LIN {X -117.613,Y -42.8309,Z 138,A -163.0883,B 24.957,C -1.5148,E1 24.85,E2 249.3615} C_DIS
LIN {X -116.0568,Y -46.8825,Z 138,A -161.1937,B 24.9576,C -1.5047,E1 24.8519,E2 247.4803} C_DIS
LIN {X -114.7173,Y -50.0725,Z 138,A -159.5986,B 24.9578,C -1.5006,E1 24.8537,E2 245.8863} C_DIS
LIN {X -112.1314,Y -55.6214,Z 138,A -156.8054,B 24.9583,C -1.4921,E1 24.857,E2 243.0981} C_DIS
LIN {X -110.6631,Y -58.4885,Z 138,A -155.2878,B 24.9584,C -1.4899,E1 24.859,E2 241.5776} C_DIS
LIN {X -108.8717,Y -61.7628,Z 138,A -153.454,B 24.9584,C -1.4909,E1 24.8615,E2 239.7318} C_DIS
LIN {X -106.6421,Y -65.5368,Z 138,A -151.0294,B 24.9576,C -1.5048,E1 24.8651,E2 237.2618} C_DIS
LIN {X -104.3746,Y -69.0914,Z 138,A -149.2788,B 24.9583,C -1.4914,E1 24.8677,E2 235.5342} C_DIS
LIN {X -102.5229,Y -71.8108,Z 138,A -148.0963,B 24.9594,C -1.4726,E1 24.8695,E2 234.3905} C_DIS
LIN {X -100.2166,Y -74.9955,Z 138,A -146.1229,B 24.9592,C -1.4761,E1 24.8728,E2 232.3994} C_DIS
LIN {X -98.095,Y -77.7497,Z 138,A -144.5728,B 24.9595,C -1.4703,E1 24.8755,E2 230.8557} C_DIS
LIN {X -95.3215,Y -81.1259,Z 138,A -142.2389,B 24.9589,C -1.4811,E1 24.8798,E2 228.4856} C_DIS
LIN {X -92.8184,Y -83.9784,Z 138,A -140.9336,B 24.9602,C -1.457,E1 24.8821,E2 227.2316} C_DIS
LIN {X -90.1766,Y -86.8095,Z 138,A -139.0349,B 24.9602,C -1.4589,E1 24.8858,E2 225.3202} C_DIS
LIN {X -87.1115,Y -89.8842,Z 138,A -137.0192,B 24.9602,C -1.456,E1 24.8898,E2 223.303} C_DIS
LIN {X -83.9565,Y -92.8382,Z 138,A -135.0831,B 24.9606,C -1.4499,E1 24.8938,E2 221.3735} C_DIS
LIN {X -80.7417,Y -95.6478,Z 138,A -132.7113,B 24.9598,C -1.4657,E1 24.8989,E2 218.955} C_DIS
LIN {X -77.6029,Y -98.2116,Z 138,A -131.2251,B 24.9609,C -1.4449,E1 24.9021,E2 217.5128} C_DIS
LIN {X -74.2065,Y -100.8017,Z 138,A -129.3231,B 24.9612,C -1.4389,E1 24.9063,E2 215.6183} C_DIS
LIN {X -70.5541,Y -103.3916,Z 138,A -127.4949,B 24.962,C -1.425,E1 24.9104,E2 213.8168} C_DIS
LIN {X -67.8733,Y -105.1709,Z 138,A -125.6046,B 24.961,C -1.4423,E1 24.9149,E2 211.8791} C_DIS
LIN {X -62.609,Y -108.3869,Z 138,A -123.181,B 24.9623,C -1.4192,E1 24.9206,E2 209.5031} C_DIS
LIN {X -59.9813,Y -109.8628,Z 138,A -121.5011,B 24.9616,C -1.4315,E1 24.9248,E2 207.7892} C_DIS
LIN {X -56.648,Y -111.616,Z 138,A -119.9096,B 24.9621,C -1.4229,E1 24.9287,E2 206.2136} C_DIS
LIN {X -53.5485,Y -113.1366,Z 138,A -118.1959,B 24.9618,C -1.4274,E1 24.9331,E2 204.485} C_DIS
LIN {X -49.8058,Y -114.8326,Z 138,A -116.3791,B 24.9621,C -1.4222,E1 24.9377,E2 202.6761} C_DIS
LIN {X -46.8573,Y -116.0669,Z 138,A -114.92,B 24.9622,C -1.4205,E1 24.9415,E2 201.2178} C_DIS
LIN {X -43.3776,Y -117.4131,Z 138,A -113.1245,B 24.9621,C -1.4231,E1 24.9462,E2 199.4124} C_DIS
LIN {X -38.9228,Y -118.9647,Z 138,A -111.1644,B 24.9627,C -1.4117,E1 24.9513,E2 197.4757} C_DIS
LIN {X -34.8619,Y -120.2161,Z 138,A -109.1765,B 24.9627,C -1.4123,E1 24.9566,E2 195.4828} C_DIS
LIN {X -31.7915,Y -121.0649,Z 138,A -107.4047,B 24.9619,C -1.4266,E1 24.9615,E2 193.6745} C_DIS
LIN {X -27.3806,Y -122.1382,Z 138,A -105.5759,B 24.9626,C -1.4134,E1 24.9664,E2 191.8746} C_DIS
LIN {X -23.6995,Y -122.9047,Z 138,A -103.8579,B 24.9626,C -1.4125,E1 24.9711,E2 190.1567} C_DIS
LIN {X -20.1619,Y -123.535,Z 138,A -102.1016,B 24.9624,C -1.4174,E1 24.976,E2 188.3871} C_DIS
LIN {X -16.1875,Y -124.1176,Z 138,A -100.4051,B 24.9628,C -1.4101,E1 24.9806,E2 186.7066} C_DIS
LIN {X -12.3645,Y -124.5573,Z 138,A -98.5723,B 24.9626,C -1.4134,E1 24.9857,E2 184.865} C_DIS
LIN {X -8.4749,Y -124.8832,Z 138,A -96.7178,B 24.9624,C -1.4166,E1 24.9909,E2 183.002} C_DIS
LIN {X -4.5423,Y -125.0869,Z 138,A -94.9814,B 24.9626,C -1.4136,E1 24.9958,E2 181.2725} C_DIS
LIN {X -0.6386,Y -125.1673,Z 138,A -93.2285,B 24.9626,C -1.4122,E1 25.0006,E2 179.5227} C_DIS
LIN {X -0.6386,Y -125.1673,Z 138,A -93.2285,B 24.9626,C -1.4122,E1 25.0006,E2 179.5227} C_DIS
Enddeposition()
LIN {X 0.8743,Y -124.1818,Z 138,A -92.728,B 24.9622,C -1.4201,E1 25.0021,E2 179.0036} C_DIS
Startdeposition()
$VEL.CP = VEL_PRINT
LIN {X -3.4324,Y -124.1396,Z 138,A -95.2903,B 24.9637,C -1.3919,E1 24.9948,E2 181.6328} C_DIS
LIN {X -7.4097,Y -123.966,Z 138,A -97.1041,B 24.9637,C -1.3929,E1 24.9897,E2 183.4448} C_DIS
LIN {X -10.9804,Y -123.7017,Z 138,A -98.832,B 24.9638,C -1.3893,E1 24.9849,E2 185.1819} C_DIS
LIN {X -14.5471,Y -123.3321,Z 138,A -100.43,B 24.9637,C -1.3922,E1 24.9804,E2 186.774} C_DIS
LIN {X -18.275,Y -122.8369,Z 138,A -102.2656,B 24.9639,C -1.3878,E1 24.9753,E2 188.6215} C_DIS
LIN {X -21.9714,Y -122.2278,Z 138,A -103.8657,B 24.9636,C -1.3945,E1 24.971,E2 190.2073} C_DIS
LIN {X -25.8177,Y -121.4741,Z 138,A -105.7547,B 24.9637,C -1.3914,E1 24.9658,E2 192.1058} C_DIS
LIN {X -30.6897,Y -120.335,Z 138,A -108.1366,B 24.9638,C -1.3892,E1 24.9593,E2 194.4961} C_DIS
LIN {X -34.3401,Y -119.3458,Z 138,A -109.8784,B 24.9638,C -1.3905,E1 24.9546,E2 196.2377} C_DIS
LIN {X -38.81,Y -117.9674,Z 138,A -111.9251,B 24.9634,C -1.3974,E1 24.9492,E2 198.2717} C_DIS
LIN {X -41.8882,Y -116.9092,Z 138,A -113.3908,B 24.9633,C -1.4004,E1 24.9453,E2 199.7331} C_DIS
LIN {X -44.8626,Y -115.8001,Z 138,A -114.8481,B 24.9632,C -1.4021,E1 24.9415,E2 201.1893} C_DIS
LIN {X -48.4333,Y -114.3543,Z 138,A -116.7893,B 24.9635,C -1.3963,E1 24.9365,E2 203.1487} C_DIS
LIN {X -51.9341,Y -112.806,Z 138,A -118.4416,B 24.9631,C -1.4037,E1 24.9323,E2 204.7876} C_DIS
LIN {X -55.0856,Y -111.3009,Z 138,A -120.0981,B 24.9631,C -1.4036,E1 24.9281,E2 206.4487} C_DIS
LIN {X -59.0081,Y -109.2743,Z 138,A -122.0954,B 24.9629,C -1.4081,E1 24.9232,E2 208.4408} C_DIS
LIN {X -62.4371,Y -107.3519,Z 138,A -123.7237,B 24.9623,C -1.4192,E1 24.9193,E2 210.0474} C_DIS
LIN {X -66.6312,Y -104.8007,Z 138,A -126.3223,B 24.9629,C -1.4073,E1 24.9131,E2 212.6825} C_DIS
LIN {X -69.5827,Y -102.864,Z 138,A -127.9674,B 24.9629,C -1.4092,E1 24.9092,E2 214.3284} C_DIS
LIN {X -72.7292,Y -100.664,Z 138,A -129.7513,B 24.9627,C -1.4116,E1 24.9052,E2 216.1127} C_DIS
LIN {X -76.3339,Y -97.9592,Z 138,A -131.9392,B 24.9627,C -1.4105,E1 24.9003,E2 218.3114} C_DIS
LIN {X -81.5463,Y -93.6642,Z 138,A -134.9089,B 24.9621,C -1.4232,E1 24.894,E2 221.2622} C_DIS
LIN {X -83.8414,Y -91.6157,Z 138,A -136.2375,B 24.9617,C -1.4302,E1 24.8913,E2 222.5795} C_DIS
LIN {X -86.675,Y -88.9401,Z 138,A -138.182,B 24.9618,C -1.4273,E1 24.8873,E2 224.5389} C_DIS
LIN {X -89.8654,Y -85.7145,Z 138,A -140.233,B 24.9615,C -1.4338,E1 24.8833,E2 226.5831} C_DIS
LIN {X -93.3293,Y -81.9299,Z 138,A -142.8298,B 24.9618,C -1.4289,E1 24.8785,E2 229.2033} C_DIS
LIN {X -96.1089,Y -78.6501,Z 138,A -144.6308,B 24.9611,C -1.4418,E1 24.8753,E2 230.9818} C_DIS
LIN {X -98.823,Y -75.212,Z 138,A -146.5442,B 24.9605,C -1.4516,E1 24.872,E2 232.8809} C_DIS
LIN {X -101.1583,Y -72.0403,Z 138,A -148.21,B 24.9599,C -1.463,E1 24.8693,E2 234.5278} C_DIS
LIN {X -103.1752,Y -69.1208,Z 138,A -150.0811,B 24.9602,C -1.4567,E1 24.8663,E2 236.423} C_DIS
LIN {X -105.8376,Y -64.9705,Z 138,A -152.385,B 24.96,C -1.4615,E1 24.8629,E2 238.7274} C_DIS
LIN {X -108.0724,Y -61.1821,Z 138,A -154.4839,B 24.9599,C -1.4639,E1 24.86,E2 240.8314} C_DIS
LIN {X -110.1847,Y -57.2875,Z 138,A -156.4851,B 24.9594,C -1.4716,E1 24.8573,E2 242.825} C_DIS
LIN {X -111.3672,Y -54.9512,Z 138,A -157.9018,B 24.9598,C -1.4658,E1 24.8556,E2 244.2632} C_DIS
LIN {X -114.2651,Y -48.6443,Z 138,A -160.9694,B 24.9589,C -1.481,E1 24.8521,E2 247.3113} C_DIS
LIN {X -115.8817,Y -44.6528,Z 138,A -162.916,B 24.9585,C -1.4887,E1 24.8501,E2 249.2504} C_DIS
LIN {X -117.2743,Y -40.8545,Z 138,A -164.6876,B 24.9579,C -1.4985,E1 24.8484,E2 251.0086} C_DIS
LIN {X -118.2722,Y -37.8684,Z 138,A -166.1592,B 24.9577,C -1.5021,E1 24.8472,E2 252.4802} C_DIS
LIN {X -119.1919,Y -34.8656,Z 138,A -167.6085,B 24.9575,C -1.5066,E1 24.846,E2 253.9272} C_DIS
LIN {X -120.1112,Y -31.5572,Z 138,A -169.2143,B 24.9573,C -1.5105,E1 24.8448,E2 255.5329} C_DIS
LIN {X -120.9616,Y -28.1224,Z 138,A -171.401,B 24.9583,C -1.4914,E1 24.8434,E2 257.7781} C_DIS
LIN {X -121.8477,Y -23.9996,Z 138,A -172.7811,B 24.9566,C -1.5223,E1 24.8427,E2 259.0927} C_DIS
LIN {X -122.5174,Y -20.2951,Z 138,A -174.9025,B 24.9572,C -1.511,E1 24.8416,E2 261.2536} C_DIS
LIN {X -123.0053,Y -17.0971,Z 138,A -176.1457,B 24.9563,C -1.5267,E1 24.8412,E2 262.4668} C_DIS
LIN {X -123.7649,Y -10.2317,Z 138,A -179.9147,B 24.9572,C -1.5116,E1 24.8401,E2 266.2942} C_DIS
LIN {X -124.0651,Y -5.5438,Z 138,A 178.388,B 24.9556,C -1.5391,E1 24.8399,E2 267.9362} C_DIS
LIN {X -124.1835,Y 1.1012,Z 138,A 174.6061,B 24.9568,C -1.5181,E1 24.8399,E2 271.7909} C_DIS
LIN {X -124.0084,Y 6.6721,Z 138,A 172.8788,B 24.9542,C -1.5632,E1 24.8401,E2 273.4211} C_DIS
LIN {X -123.3586,Y 14.3242,Z 138,A 168.7788,B 24.955,C -1.5506,E1 24.8412,E2 277.5759} C_DIS
LIN {X -122.8256,Y 18.3457,Z 138,A 167.1473,B 24.954,C -1.5671,E1 24.8418,E2 279.1777} C_DIS
LIN {X -122.3011,Y 21.562,Z 138,A 164.8552,B 24.9557,C -1.538,E1 24.843,E2 281.5529} C_DIS
LIN {X -121.0008,Y 27.9507,Z 138,A 162.7356,B 24.9529,C -1.5861,E1 24.8442,E2 283.5701} C_DIS
LIN {X -119.9687,Y 32.0913,Z 138,A 160.8421,B 24.9523,C -1.5958,E1 24.8455,E2 285.4516} C_DIS
LIN {X -118.9059,Y 35.8329,Z 138,A 159.0623,B 24.9519,C -1.6022,E1 24.8469,E2 287.2265} C_DIS
LIN {X -117.8267,Y 39.2325,Z 138,A 157.3944,B 24.9516,C -1.6064,E1 24.8484,E2 288.8938} C_DIS
LIN {X -116.6428,Y 42.6269,Z 138,A 155.6155,B 24.9516,C -1.6064,E1 24.85,E2 290.6829} C_DIS
LIN {X -114.779,Y 47.4161,Z 138,A 153.2191,B 24.9513,C -1.6127,E1 24.8525,E2 293.0776} C_DIS
LIN {X -112.351,Y 52.9151,Z 138,A 150.4157,B 24.9508,C -1.6199,E1 24.8557,E2 295.8793} C_DIS
LIN {X -110.5037,Y 56.6688,Z 138,A 148.0759,B 24.9516,C -1.6078,E1 24.8588,E2 298.2603} C_DIS
LIN {X -108.4775,Y 60.4608,Z 138,A 146.8277,B 24.9492,C -1.6459,E1 24.8603,E2 299.4244} C_DIS
LIN {X -105.5316,Y 65.4665,Z 138,A 143.8039,B 24.9497,C -1.6385,E1 24.8647,E2 302.4814} C_DIS
LIN {X -103.3904,Y 68.7983,Z 138,A 141.9856,B 24.9493,C -1.6441,E1 24.8675,E2 304.2954} C_DIS
LIN {X -100.9087,Y 72.3894,Z 138,A 140.0193,B 24.9489,C -1.6519,E1 24.8706,E2 306.253} C_DIS
LIN {X -98.4124,Y 75.7489,Z 138,A 137.9685,B 24.9489,C -1.6519,E1 24.8741,E2 308.3137} C_DIS
LIN {X -95.6749,Y 79.1774,Z 138,A 136.0126,B 24.9483,C -1.6603,E1 24.8775,E2 310.2585} C_DIS
LIN {X -92.9507,Y 82.3586,Z 138,A 134.074,B 24.948,C -1.6651,E1 24.881,E2 312.1946} C_DIS
LIN {X -90.1146,Y 85.453,Z 138,A 132.0632,B 24.948,C -1.6667,E1 24.8849,E2 314.2104} C_DIS
LIN {X -87.1027,Y 88.5206,Z 138,A 130.0953,B 24.9476,C -1.6722,E1 24.8887,E2 316.1734} C_DIS
LIN {X -84.0026,Y 91.4675,Z 138,A 128.1473,B 24.9472,C -1.6781,E1 24.8927,E2 318.1154} C_DIS
LIN {X -80.7834,Y 94.3234,Z 138,A 126.0842,B 24.9472,C -1.6792,E1 24.8971,E2 320.1839} C_DIS
LIN {X -77.485,Y 97.0508,Z 138,A 124.1423,B 24.9468,C -1.6851,E1 24.9012,E2 322.1192} C_DIS
LIN {X -74.2978,Y 99.5119,Z 138,A 122.2503,B 24.9466,C -1.6875,E1 24.9055,E2 324.0123} C_DIS
LIN {X -70.7447,Y 102.0685,Z 138,A 120.2293,B 24.9464,C -1.6916,E1 24.9101,E2 326.0306} C_DIS
LIN {X -67.2251,Y 104.4205,Z 138,A 118.2372,B 24.9462,C -1.6937,E1 24.9147,E2 328.0242} C_DIS
LIN {X -64.3323,Y 106.2267,Z 138,A 116.8746,B 24.9454,C -1.7061,E1 24.9179,E2 329.3614} C_DIS
LIN {X -59.0981,Y 109.2259,Z 138,A 113.8547,B 24.9458,C -1.7004,E1 24.9253,E2 332.4038} C_DIS
LIN {X -56.1772,Y 110.754,Z 138,A 111.8837,B 24.9469,C -1.6827,E1 24.9303,E2 334.4221} C_DIS
LIN {X -52.1747,Y 112.6947,Z 138,A 110.3031,B 24.9454,C -1.7072,E1 24.9342,E2 335.9486} C_DIS
LIN {X -48.2211,Y 114.4429,Z 138,A 108.4908,B 24.9447,C -1.7184,E1 24.9388,E2 337.7384} C_DIS
LIN {X -45.1901,Y 115.6728,Z 138,A 106.8881,B 24.9447,C -1.7162,E1 24.9429,E2 339.3498} C_DIS
LIN {X -42.1787,Y 116.8044,Z 138,A 104.7649,B 24.9465,C -1.6892,E1 24.9487,E2 341.5415} C_DIS
LIN {X -37.7002,Y 118.3259,Z 138,A 103.2224,B 24.9445,C -1.7209,E1 24.9526,E2 343.0115} C_DIS
LIN {X -34.1667,Y 119.3965,Z 138,A 101.4889,B 24.9445,C -1.7214,E1 24.9572,E2 344.7468} C_DIS
LIN {X -30.834,Y 120.2984,Z 138,A 99.836,B 24.9445,C -1.7203,E1 24.9617,E2 346.4047} C_DIS
LIN {X -26.292,Y 121.3717,Z 138,A 97.4667,B 24.9451,C -1.7123,E1 24.9682,E2 348.7959} C_DIS
LIN {X -21.4393,Y 122.323,Z 138,A 95.3635,B 24.9444,C -1.7223,E1 24.974,E2 350.8776} C_DIS
LIN {X -17.5315,Y 122.9432,Z 138,A 93.611,B 24.9441,C -1.727,E1 24.9788,E2 352.6206} C_DIS
LIN {X -13.9053,Y 123.4075,Z 138,A 91.9272,B 24.9441,C -1.728,E1 24.9834,E2 354.303} C_DIS
LIN {X -10.5557,Y 123.7376,Z 138,A 90.3559,B 24.9441,C -1.728,E1 24.9878,E2 355.8752} C_DIS
LIN {X -6.4421,Y 124.02,Z 138,A 88.4669,B 24.944,C -1.7294,E1 24.9931,E2 357.7616} C_DIS
LIN {X -2.553,Y 124.1618,Z 138,A 86.6125,B 24.944,C -1.7271,E1 24.9982,E2 359.6216} C_DIS
LIN {X 1.5275,Y 124.1788,Z 138,A 84.718,B 24.9441,C -1.7269,E1 25.0035,E2 361.5164} C_DIS
LIN {X 5.5023,Y 124.0668,Z 138,A 82.8509,B 24.9442,C -1.7255,E1 25.0088,E2 363.3863} C_DIS
LIN {X 9.4083,Y 123.8306,Z 138,A 81.078,B 24.9442,C -1.727,E1 25.0137,E2 365.1549} C_DIS
LIN {X 13.3038,Y 123.4723,Z 138,A 79.3529,B 24.9439,C -1.7305,E1 25.0185,E2 366.8706} C_DIS
LIN {X 17.2613,Y 122.9818,Z 138,A 77.5039,B 24.9439,C -1.7297,E1 25.0236,E2 368.7201} C_DIS
LIN {X 20.2718,Y 122.5212,Z 138,A 76.1293,B 24.9439,C -1.7307,E1 25.0274,E2 370.091} C_DIS
LIN {X 23.7432,Y 121.8967,Z 138,A 74.6464,B 24.9435,C -1.7369,E1 25.0314,E2 371.5575} C_DIS
LIN {X 28.228,Y 120.9375,Z 138,A 72.2634,B 24.9444,C -1.723,E1 25.038,E2 373.9701} C_DIS
LIN {X 34.0853,Y 119.4191,Z 138,A 69.5144,B 24.9444,C -1.7232,E1 25.0454,E2 376.7144} C_DIS
LIN {X 37.5407,Y 118.3769,Z 138,A 67.9097,B 24.9442,C -1.7248,E1 25.0496,E2 378.3123} C_DIS
LIN {X 40.6961,Y 117.3292,Z 138,A 66.5544,B 24.9438,C -1.7321,E1 25.0532,E2 379.6478} C_DIS
LIN {X 43.2115,Y 116.4268,Z 138,A 65.1953,B 24.9442,C -1.7249,E1 25.0568,E2 381.0212} C_DIS
LIN {X 47.2977,Y 114.8286,Z 138,A 63.0652,B 24.9447,C -1.7176,E1 25.0623,E2 383.1636} C_DIS
LIN {X 50.5904,Y 113.4148,Z 138,A 61.4843,B 24.9447,C -1.7193,E1 25.0663,E2 384.7367} C_DIS
LIN {X 55.029,Y 111.3288,Z 138,A 59.2396,B 24.9447,C -1.7174,E1 25.072,E2 386.9801} C_DIS
LIN {X 58.3696,Y 109.6166,Z 138,A 57.4755,B 24.945,C -1.7134,E1 25.0764,E2 388.7485} C_DIS
LIN {X 63.9806,Y 106.4394,Z 138,A 54.4267,B 24.9455,C -1.7055,E1 25.0838,E2 391.8071} C_DIS
LIN {X 66.9888,Y 104.5718,Z 138,A 53.0523,B 24.9448,C -1.7156,E1 25.087,E2 393.1532} C_DIS
LIN {X 69.9022,Y 102.6477,Z 138,A 51.1942,B 24.9458,C -1.7008,E1 25.0913,E2 395.04} C_DIS
LIN {X 73.4675,Y 100.1263,Z 138,A 49.244,B 24.9458,C -1.7004,E1 25.0957,E2 396.9843} C_DIS
LIN {X 76.9488,Y 97.4768,Z 138,A 47.1956,B 24.9461,C -1.6952,E1 25.1003,E2 399.0375} C_DIS
LIN {X 80.1244,Y 94.8841,Z 138,A 45.287,B 24.9464,C -1.6907,E1 25.1044,E2 400.9494} C_DIS
LIN {X 83.4378,Y 91.9831,Z 138,A 43.2992,B 24.9466,C -1.6887,E1 25.1085,E2 402.9339} C_DIS
LIN {X 86.9726,Y 88.6483,Z 138,A 41.0769,B 24.9468,C -1.6849,E1 25.113,E2 405.1559} C_DIS
LIN {X 89.9625,Y 85.6129,Z 138,A 39.0959,B 24.9471,C -1.6798,E1 25.1168,E2 407.1405} C_DIS
LIN {X 92.246,Y 83.1479,Z 138,A 37.5275,B 24.9474,C -1.6753,E1 25.1198,E2 408.7125} C_DIS
LIN {X 95.1662,Y 79.7881,Z 138,A 35.5789,B 24.9474,C -1.6757,E1 25.1233,E2 410.6514} C_DIS
LIN {X 97.7814,Y 76.561,Z 138,A 33.6191,B 24.9478,C -1.6689,E1 25.1267,E2 412.6182} C_DIS
LIN {X 100.4007,Y 73.0926,Z 138,A 31.5508,B 24.9483,C -1.6607,E1 25.1302,E2 414.6959} C_DIS
LIN {X 103.0668,Y 69.2824,Z 138,A 29.5462,B 24.9483,C -1.6622,E1 25.1334,E2 416.6871} C_DIS
LIN {X 105.2347,Y 65.9436,Z 138,A 27.6161,B 24.9488,C -1.6526,E1 25.1363,E2 418.63} C_DIS
LIN {X 106.9997,Y 63.0385,Z 138,A 26.046,B 24.9491,C -1.6482,E1 25.1385,E2 420.2024} C_DIS
LIN {X 109.2222,Y 59.1051,Z 138,A 23.9718,B 24.9494,C -1.643,E1 25.1413,E2 422.2782} C_DIS
LIN {X 110.8631,Y 55.9628,Z 138,A 21.883,B 24.9511,C -1.6156,E1 25.144,E2 424.4202} C_DIS
LIN {X 112.8849,Y 51.7635,Z 138,A 20.2307,B 24.9499,C -1.6344,E1 25.1459,E2 426.0194} C_DIS
LIN {X 114.5193,Y 48.0383,Z 138,A 18.494,B 24.9499,C -1.636,E1 25.1478,E2 427.7429} C_DIS
LIN {X 115.6403,Y 45.2738,Z 138,A 17.0947,B 24.9502,C -1.6307,E1 25.1492,E2 429.1469} C_DIS
LIN {X 116.8385,Y 42.0842,Z 138,A 15.5809,B 24.9502,C -1.6289,E1 25.1507,E2 430.6565} C_DIS
LIN {X 119.168,Y 34.9474,Z 138,A 11.7607,B 24.952,C -1.6002,E1 25.154,E2 434.5225} C_DIS
LIN {X 120.107,Y 31.5728,Z 138,A 10.5006,B 24.9512,C -1.6132,E1 25.1548,E2 435.7449} C_DIS
LIN {X 121.585,Y 25.2931,Z 138,A 7.5126,B 24.9518,C -1.6032,E1 25.1567,E2 438.7391} C_DIS
LIN {X 122.1968,Y 22.1447,Z 138,A 6.1154,B 24.9518,C -1.6027,E1 25.1574,E2 440.1293} C_DIS
LIN {X 122.7491,Y 18.843,Z 138,A 4.5465,B 24.9522,C -1.5965,E1 25.1581,E2 441.7037} C_DIS
LIN {X 123.2945,Y 14.862,Z 138,A 2.709,B 24.9526,C -1.5913,E1 25.1588,E2 443.5424} C_DIS
LIN {X 123.6905,Y 11.1134,Z 138,A 0.8636,B 24.9532,C -1.5802,E1 25.1593,E2 445.4031} C_DIS
LIN {X 123.9807,Y 7.1706,Z 138,A -0.9361,B 24.9535,C -1.5755,E1 25.1596,E2 447.2032} C_DIS
LIN {X 124.148,Y 3.1299,Z 138,A -2.7111,B 24.9535,C -1.574,E1 25.1598,E2 448.9712} C_DIS
LIN {X 124.1867,Y -0.6774,Z 138,A -4.5473,B 24.9542,C -1.5642,E1 25.1598,E2 450.8196} C_DIS
LIN {X 124.0912,Y -4.8766,Z 138,A -6.3646,B 24.9542,C -1.564,E1 25.1596,E2 452.6266} C_DIS
LIN {X 123.8774,Y -8.7669,Z 138,A -8.1646,B 24.9545,C -1.5579,E1 25.1593,E2 454.4302} C_DIS
LIN {X 123.5541,Y -12.5391,Z 138,A -9.9033,B 24.9548,C -1.5525,E1 25.1589,E2 456.1712} C_DIS
LIN {X 123.1453,Y -16.0506,Z 138,A -11.5168,B 24.9551,C -1.5481,E1 25.1583,E2 457.7857} C_DIS
LIN {X 122.5421,Y -20.1466,Z 138,A -13.3482,B 24.9552,C -1.5459,E1 25.1575,E2 459.6116} C_DIS
LIN {X 121.978,Y -23.3178,Z 138,A -14.7926,B 24.9554,C -1.5431,E1 25.1568,E2 461.0539} C_DIS
LIN {X 120.2902,Y -30.866,Z 138,A -18.4532,B 24.9563,C -1.5268,E1 25.1545,E2 464.7319} C_DIS
LIN {X 118.2301,Y -38.0001,Z 138,A -21.8267,B 24.9568,C -1.5184,E1 25.1518,E2 468.1058} C_DIS
LIN {X 116.5846,Y -42.7885,Z 138,A -24.2446,B 24.9575,C -1.5068,E1 25.1496,E2 470.5376} C_DIS
LIN {X 115.1834,Y -46.423,Z 138,A -25.8147,B 24.9571,C -1.5128,E1 25.148,E2 472.0849} C_DIS
LIN {X 113.9184,Y -49.4461,Z 138,A -27.7895,B 24.9587,C -1.4845,E1 25.1457,E2 474.1154} C_DIS
LIN {X 112.4177,Y -52.7737,Z 138,A -29.2005,B 24.9582,C -1.4931,E1 25.1441,E2 475.4984} C_DIS
LIN {X 110.7688,Y -56.1481,Z 138,A -30.8076,B 24.9582,C -1.4943,E1 25.1421,E2 477.0942} C_DIS
LIN {X 108.9163,Y -59.6661,Z 138,A -32.7379,B 24.9587,C -1.4839,E1 25.1396,E2 479.039} C_DIS
LIN {X 106.8177,Y -63.3468,Z 138,A -34.6805,B 24.959,C -1.4787,E1 25.1368,E2 480.9837} C_DIS
LIN {X 104.422,Y -67.2227,Z 138,A -36.7615,B 24.9593,C -1.4737,E1 25.1337,E2 483.0661} C_DIS
LIN {X 102.1043,Y -70.6933,Z 138,A -38.6668,B 24.9596,C -1.4692,E1 25.1307,E2 484.9724} C_DIS
LIN {X 99.8317,Y -73.8683,Z 138,A -40.2974,B 24.9594,C -1.4729,E1 25.1281,E2 486.5867} C_DIS
LIN {X 97.2143,Y -77.2797,Z 138,A -42.1733,B 24.9594,C -1.4729,E1 25.1249,E2 488.4535} C_DIS
LIN {X 95.4684,Y -79.4268,Z 138,A -43.7078,B 24.9603,C -1.4564,E1 25.1221,E2 490.0199} C_DIS
LIN {X 92.733,Y -82.6042,Z 138,A -45.5919,B 24.9604,C -1.4539,E1 25.1187,E2 491.9015} C_DIS
LIN {X 88.9481,Y -86.6668,Z 138,A -48.2579,B 24.961,C -1.4421,E1 25.1135,E2 494.5837} C_DIS
LIN {X 85.6338,Y -89.9425,Z 138,A -50.3072,B 24.961,C -1.4419,E1 25.1094,E2 496.6249} C_DIS
LIN {X 82.529,Y -92.8,Z 138,A -52.5342,B 24.9621,C -1.4232,E1 25.1047,E2 498.887} C_DIS
LIN {X 79.8918,Y -95.0792,Z 138,A -54.0398,B 24.962,C -1.4247,E1 25.1015,E2 500.3834} C_DIS
LIN {X 75.9842,Y -98.2302,Z 138,A -56.0862,B 24.9615,C -1.433,E1 25.0971,E2 502.4025} C_DIS
LIN {X 73.1125,Y -100.3863,Z 138,A -57.8088,B 24.9619,C -1.4262,E1 25.0932,E2 504.1351} C_DIS
LIN {X 67.3884,Y -104.3151,Z 138,A -60.9996,B 24.9622,C -1.4203,E1 25.0858,E2 507.3291} C_DIS
LIN {X 63.7638,Y -106.5691,Z 138,A -62.6925,B 24.9617,C -1.4303,E1 25.0819,E2 508.993} C_DIS
LIN {X 61.3937,Y -107.9517,Z 138,A -64.6519,B 24.9636,C -1.3936,E1 25.0769,E2 511.0333} C_DIS
LIN {X 57.7626,Y -109.9353,Z 138,A -65.9935,B 24.9623,C -1.4183,E1 25.0738,E2 512.3126} C_DIS
LIN {X 54.9367,Y -111.3744,Z 138,A -67.4652,B 24.9625,C -1.4154,E1 25.0701,E2 513.7872} C_DIS
LIN {X 51.8939,Y -112.8246,Z 138,A -69.0579,B 24.9627,C -1.4111,E1 25.066,E2 515.3861} C_DIS
LIN {X 48.0729,Y -114.5048,Z 138,A -70.9707,B 24.9628,C -1.4088,E1 25.0611,E2 517.2997} C_DIS
LIN {X 45.2613,Y -115.6452,Z 138,A -72.3349,B 24.9628,C -1.4085,E1 25.0576,E2 518.6614} C_DIS
LIN {X 39.9764,Y -117.5787,Z 138,A -74.9025,B 24.9629,C -1.4064,E1 25.0509,E2 521.2287} C_DIS
LIN {X 33.4884,Y -119.5862,Z 138,A -78.2116,B 24.9636,C -1.3942,E1 25.0419,E2 524.5609} C_DIS
LIN {X 30.4141,Y -120.4049,Z 138,A -79.7975,B 24.964,C -1.3869,E1 25.0376,E2 526.1617} C_DIS
LIN {X 23.8034,Y -121.8852,Z 138,A -82.7546,B 24.9637,C -1.3922,E1 25.0296,E2 529.1025} C_DIS
LIN {X 19.5737,Y -122.636,Z 138,A -84.7032,B 24.9637,C -1.3922,E1 25.0242,E2 531.0489} C_DIS
LIN {X 15.7542,Y -123.1842,Z 138,A -86.3934,B 24.9635,C -1.3955,E1 25.0196,E2 532.7301} C_DIS
LIN {X 12.3548,Y -123.5718,Z 138,A -88.0742,B 24.9638,C -1.3896,E1 25.0149,E2 534.4236} C_DIS
LIN {X 8.2171,Y -123.9162,Z 138,A -89.9919,B 24.9638,C -1.3886,E1 25.0095,E2 536.3428} C_DIS
LIN {X 4.2625,Y -124.1152,Z 138,A -91.8055,B 24.9638,C -1.3886,E1 25.0045,E2 538.1561} C_DIS
LIN {X 0.8743,Y -124.1818,Z 138,A -92.7259,B 24.9623,C -1.4192,E1 25.0021,E2 539.0036} C_DIS
Enddeposition()
LIN {X 0.8743,Y -124.1818,Z 138,A -92.7259,B 24.9623,C -1.4192,E1 25.0021,E2 539.0036} C_DIS
Startdeposition()
$VEL.CP = VEL_PRINT
LIN {X 2.906,Y -123.172,Z 138,A -91.5342,B 24.7909,C -1.4123,E1 24.834,E2 537.804} C_DIS
LIN {X 6.8533,Y -123.0162,Z 138,A -89.635,B 24.7907,C -1.416,E1 24.8393,E2 535.8966} C_DIS
LIN {X 10.7412,Y -122.7365,Z 138,A -87.8538,B 24.7907,C -1.4154,E1 24.8443,E2 534.1178} C_DIS
LIN {X 14.115,Y -122.3948,Z 138,A -86.327,B 24.7908,C -1.4139,E1 24.8485,E2 532.5957} C_DIS
LIN {X 17.7325,Y -121.9226,Z 138,A -84.5753,B 24.7906,C -1.4178,E1 24.8534,E2 530.8364} C_DIS
LIN {X 21.363,Y -121.3392,Z 138,A -82.9343,B 24.7907,C -1.4157,E1 24.8579,E2 529.2019} C_DIS
LIN {X 24.666,Y -120.7106,Z 138,A -80.7554,B 24.789,C -1.4473,E1 24.864,E2 526.9507} C_DIS
LIN {X 29.5588,Y -119.6086,Z 138,A -79.0093,B 24.7905,C -1.4207,E1 24.8686,E2 525.2703} C_DIS
LIN {X 33.0399,Y -118.6921,Z 138,A -77.6285,B 24.7911,C -1.4083,E1 24.8722,E2 523.9214} C_DIS
LIN {X 38.6221,Y -116.9951,Z 138,A -74.648,B 24.7903,C -1.4245,E1 24.8803,E2 520.9076} C_DIS
LIN {X 41.2597,Y -116.092,Z 138,A -73.216,B 24.7898,C -1.4329,E1 24.8841,E2 519.4587} C_DIS
LIN {X 45.4135,Y -114.5317,Z 138,A -71.4335,B 24.7904,C -1.4219,E1 24.8886,E2 517.7063} C_DIS
LIN {X 48.7058,Y -113.1688,Z 138,A -69.8827,B 24.7905,C -1.4191,E1 24.8926,E2 516.1656} C_DIS
LIN {X 51.6272,Y -111.8661,Z 138,A -68.1438,B 24.7897,C -1.4339,E1 24.8971,E2 514.3961} C_DIS
LIN {X 55.6627,Y -109.9141,Z 138,A -66.0561,B 24.7896,C -1.4375,E1 24.9023,E2 512.3055} C_DIS
LIN {X 62.9853,Y -105.8901,Z 138,A -62.197,B 24.7892,C -1.4431,E1 24.9117,E2 508.4445} C_DIS
LIN {X 66.6373,Y -103.6309,Z 138,A -60.335,B 24.7894,C -1.4402,E1 24.9161,E2 506.5953} C_DIS
LIN {X 70.1898,Y -101.2585,Z 138,A -58.3468,B 24.7892,C -1.4443,E1 24.9207,E2 504.6041} C_DIS
LIN {X 73.1736,Y -99.1239,Z 138,A -56.5474,B 24.7887,C -1.4526,E1 24.9248,E2 502.7914} C_DIS
LIN {X 76.175,Y -96.8361,Z 138,A -54.7987,B 24.7885,C -1.4561,E1 24.9287,E2 501.0409} C_DIS
LIN {X 78.8355,Y -94.6833,Z 138,A -53.3498,B 24.7887,C -1.4526,E1 24.9318,E2 499.6059} C_DIS
LIN {X 81.6434,Y -92.2724,Z 138,A -51.4918,B 24.7881,C -1.4635,E1 24.9357,E2 497.7295} C_DIS
LIN {X 84.701,Y -89.4741,Z 138,A -49.5798,B 24.7879,C -1.4673,E1 24.9396,E2 495.8162} C_DIS
LIN {X 87.5953,Y -86.6428,Z 138,A -47.7194,B 24.7877,C -1.4708,E1 24.9433,E2 493.9554} C_DIS
LIN {X 90.6105,Y -83.4841,Z 138,A -45.6835,B 24.7874,C -1.4763,E1 24.9472,E2 491.9155} C_DIS
LIN {X 93.4728,Y -80.2665,Z 138,A -43.6941,B 24.7872,C -1.4808,E1 24.9509,E2 489.9243} C_DIS
LIN {X 96.1203,Y -77.0769,Z 138,A -41.8747,B 24.7872,C -1.4805,E1 24.9541,E2 488.1141} C_DIS
LIN {X 98.4433,Y -74.0863,Z 138,A -40.018,B 24.7866,C -1.4902,E1 24.9572,E2 486.2433} C_DIS
LIN {X 100.5569,Y -71.1913,Z 138,A -38.372,B 24.7864,C -1.4938,E1 24.9599,E2 484.5968} C_DIS
LIN {X 102.9725,Y -67.6499,Z 138,A -36.4077,B 24.7862,C -1.498,E1 24.963,E2 482.6323} C_DIS
LIN {X 105.1576,Y -64.2012,Z 138,A -34.4963,B 24.7858,C -1.5042,E1 24.9658,E2 480.7161} C_DIS
LIN {X 107.2123,Y -60.7084,Z 138,A -32.6423,B 24.7856,C -1.5082,E1 24.9684,E2 478.8623} C_DIS
LIN {X 110.1554,Y -55.1882,Z 138,A -29.8566,B 24.7855,C -1.5107,E1 24.972,E2 476.0856} C_DIS
LIN {X 113.5259,Y -47.8691,Z 138,A -26.0972,B 24.7848,C -1.5227,E1 24.9763,E2 472.3181} C_DIS
LIN {X 114.6058,Y -45.2251,Z 138,A -24.675,B 24.7843,C -1.5317,E1 24.9778,E2 470.8826} C_DIS
LIN {X 115.9586,Y -41.6299,Z 138,A -22.9438,B 24.7841,C -1.5345,E1 24.9794,E2 469.1544} C_DIS
LIN {X 117.3729,Y -37.4569,Z 138,A -20.7194,B 24.7832,C -1.55,E1 24.9814,E2 466.9059} C_DIS
LIN {X 118.6351,Y -33.2438,Z 138,A -18.9315,B 24.7836,C -1.5434,E1 24.9828,E2 465.1439} C_DIS
LIN {X 119.5254,Y -29.8883,Z 138,A -17.3437,B 24.7834,C -1.5473,E1 24.9839,E2 463.5562} C_DIS
LIN {X 120.2504,Y -26.827,Z 138,A -15.5022,B 24.7819,C -1.5714,E1 24.985,E2 461.6683} C_DIS
LIN {X 120.9517,Y -23.4576,Z 138,A -14.2489,B 24.7827,C -1.5588,E1 24.9857,E2 460.4522} C_DIS
LIN {X 121.5911,Y -19.8806,Z 138,A -12.5433,B 24.7823,C -1.5651,E1 24.9865,E2 458.7417} C_DIS
LIN {X 122.1887,Y -15.7936,Z 138,A -10.6233,B 24.7819,C -1.5714,E1 24.9872,E2 456.8183} C_DIS
LIN {X 122.6381,Y -11.806,Z 138,A -8.8849,B 24.7819,C -1.571,E1 24.9877,E2 455.0911} C_DIS
LIN {X 122.9215,Y -8.376,Z 138,A -7.152,B 24.7812,C -1.583,E1 24.9881,E2 453.3402} C_DIS
LIN {X 123.1242,Y -4.4783,Z 138,A -5.3537,B 24.7809,C -1.5881,E1 24.9883,E2 451.5404} C_DIS
LIN {X 123.2076,Y -0.2312,Z 138,A -3.4194,B 24.7807,C -1.5925,E1 24.9883,E2 449.6074} C_DIS
LIN {X 123.1574,Y 3.4316,Z 138,A -1.7838,B 24.7805,C -1.5947,E1 24.9883,E2 447.9765} C_DIS
LIN {X 122.9804,Y 7.4393,Z 138,A -0.0451,B 24.7805,C -1.5943,E1 24.988,E2 446.2492} C_DIS
LIN {X 122.7652,Y 10.4023,Z 138,A 1.44,B 24.78,C -1.6041,E1 24.9877,E2 444.7497} C_DIS
LIN {X 122.346,Y 14.5239,Z 138,A 3.3765,B 24.7796,C -1.6108,E1 24.9871,E2 442.8088} C_DIS
LIN {X 121.7854,Y 18.65,Z 138,A 5.2637,B 24.7793,C -1.6145,E1 24.9863,E2 440.924} C_DIS
LIN {X 121.1384,Y 22.4811,Z 138,A 7.1576,B 24.7787,C -1.6247,E1 24.9854,E2 439.0172} C_DIS
LIN {X 119.8367,Y 28.6125,Z 138,A 10.0277,B 24.7783,C -1.6316,E1 24.9837,E2 436.1474} C_DIS
LIN {X 118.8015,Y 32.6489,Z 138,A 11.9196,B 24.7781,C -1.6353,E1 24.9823,E2 434.2577} C_DIS
LIN {X 116.6645,Y 39.6148,Z 138,A 15.3773,B 24.7772,C -1.6491,E1 24.9794,E2 430.787} C_DIS
LIN {X 115.5464,Y 42.7628,Z 138,A 16.629,B 24.7779,C -1.6386,E1 24.9782,E2 429.5674} C_DIS
LIN {X 114.348,Y 45.8692,Z 138,A 18.3382,B 24.7771,C -1.6513,E1 24.9765,E2 427.8376} C_DIS
LIN {X 113.0968,Y 48.8723,Z 138,A 19.7795,B 24.7771,C -1.6521,E1 24.9749,E2 426.4022} C_DIS
LIN {X 111.9515,Y 51.4425,Z 138,A 21.2368,B 24.7763,C -1.6634,E1 24.9732,E2 424.9261} C_DIS
LIN {X 110.0551,Y 55.3858,Z 138,A 23.2266,B 24.7761,C -1.6669,E1 24.9707,E2 422.9387} C_DIS
LIN {X 108.4293,Y 58.5063,Z 138,A 24.8302,B 24.7759,C -1.6698,E1 24.9686,E2 421.3367} C_DIS
LIN {X 106.8163,Y 61.4025,Z 138,A 26.452,B 24.7754,C -1.6781,E1 24.9664,E2 419.7038} C_DIS
LIN {X 104.3967,Y 65.4318,Z 138,A 28.5775,B 24.7752,C -1.681,E1 24.9633,E2 417.5824} C_DIS
LIN {X 102.4394,Y 68.4545,Z 138,A 30.2171,B 24.775,C -1.6836,E1 24.9608,E2 415.9447} C_DIS
LIN {X 98.6995,Y 73.7448,Z 138,A 33.2252,B 24.7746,C -1.691,E1 24.9559,E2 412.9338} C_DIS
LIN {X 96.1394,Y 77.0532,Z 138,A 35.2013,B 24.7742,C -1.6973,E1 24.9524,E2 410.9521} C_DIS
LIN {X 93.313,Y 80.4521,Z 138,A 37.1487,B 24.7742,C -1.6968,E1 24.9489,E2 409.0149} C_DIS
LIN {X 90.571,Y 83.5271,Z 138,A 39.0318,B 24.774,C -1.6995,E1 24.9454,E2 407.1337} C_DIS
LIN {X 87.7648,Y 86.4712,Z 138,A 41.0071,B 24.7735,C -1.7079,E1 24.9415,E2 405.1471} C_DIS
LIN {X 84.5577,Y 89.6094,Z 138,A 43.0632,B 24.7733,C -1.7108,E1 24.9374,E2 403.0926} C_DIS
LIN {X 81.5083,Y 92.3918,Z 138,A 44.9699,B 24.7731,C -1.7141,E1 24.9334,E2 401.1858} C_DIS
LIN {X 78.3484,Y 95.0866,Z 138,A 46.9282,B 24.7727,C -1.7192,E1 24.9292,E2 399.2231} C_DIS
LIN {X 75.234,Y 97.5694,Z 138,A 48.6449,B 24.7729,C -1.7159,E1 24.9255,E2 397.5204} C_DIS
LIN {X 72.2552,Y 99.7949,Z 138,A 50.4367,B 24.7725,C -1.7221,E1 24.9214,E2 395.7204} C_DIS
LIN {X 68.9944,Y 102.0766,Z 138,A 52.662,B 24.7711,C -1.7436,E1 24.9162,E2 393.4515} C_DIS
LIN {X 65.853,Y 104.1309,Z 138,A 54.064,B 24.7721,C -1.7295,E1 24.913,E2 392.0875} C_DIS
LIN {X 62.5323,Y 106.1583,Z 138,A 55.9858,B 24.7715,C -1.7378,E1 24.9084,E2 390.1522} C_DIS
LIN {X 58.9502,Y 108.1884,Z 138,A 57.6327,B 24.7722,C -1.7274,E1 24.9044,E2 388.5347} C_DIS
LIN {X 56.0633,Y 109.7102,Z 138,A 59.0944,B 24.7722,C -1.7268,E1 24.9008,E2 387.0787} C_DIS
LIN {X 53.2068,Y 111.1235,Z 138,A 60.5536,B 24.7722,C -1.7276,E1 24.8971,E2 385.6215} C_DIS
LIN {X 50.4596,Y 112.3977,Z 138,A 62.0837,B 24.7717,C -1.7351,E1 24.8932,E2 384.0774} C_DIS
LIN {X 46.6274,Y 114.0424,Z 138,A 64.1326,B 24.7712,C -1.7425,E1 24.8879,E2 382.0158} C_DIS
LIN {X 42.4809,Y 115.6518,Z 138,A 66.0352,B 24.7716,C -1.7365,E1 24.883,E2 380.1315} C_DIS
LIN {X 38.9848,Y 116.8743,Z 138,A 67.7155,B 24.7716,C -1.736,E1 24.8786,E2 378.4557} C_DIS
LIN {X 34.7779,Y 118.1946,Z 138,A 69.7534,B 24.7716,C -1.737,E1 24.8731,E2 376.4191} C_DIS
LIN {X 29.6762,Y 119.5792,Z 138,A 72.4303,B 24.7708,C -1.749,E1 24.8658,E2 373.7179} C_DIS
LIN {X 26.7662,Y 120.2642,Z 138,A 74.0786,B 24.7699,C -1.762,E1 24.8613,E2 372.0407} C_DIS
LIN {X 23.4015,Y 120.9624,Z 138,A 75.3493,B 24.7709,C -1.7471,E1 24.8579,E2 370.8071} C_DIS
LIN {X 19.2621,Y 121.6906,Z 138,A 77.2992,B 24.7709,C -1.7476,E1 24.8525,E2 368.8581} C_DIS
LIN {X 15.6283,Y 122.2104,Z 138,A 79.0737,B 24.7706,C -1.7512,E1 24.8476,E2 367.0765} C_DIS
LIN {X 12.1719,Y 122.603,Z 138,A 80.5251,B 24.7711,C -1.7436,E1 24.8436,E2 365.6442} C_DIS
LIN {X 8.8135,Y 122.8896,Z 138,A 82.2311,B 24.7707,C -1.7502,E1 24.8388,E2 363.9233} C_DIS
LIN {X 4.7695,Y 123.1128,Z 138,A 84.0314,B 24.771,C -1.7462,E1 24.8338,E2 362.133} C_DIS
LIN {X 0.8921,Y 123.2022,Z 138,A 85.8899,B 24.7708,C -1.7485,E1 24.8286,E2 360.2693} C_DIS
LIN {X -3.4229,Y 123.1576,Z 138,A 87.895,B 24.7708,C -1.7479,E1 24.823,E2 358.2655} C_DIS
LIN {X -7.471,Y 122.9784,Z 138,A 89.7256,B 24.7711,C -1.7447,E1 24.8179,E2 356.442} C_DIS
LIN {X -11.195,Y 122.6968,Z 138,A 91.5341,B 24.7709,C -1.7472,E1 24.8129,E2 354.6266} C_DIS
LIN {X -15.0775,Y 122.28,Z 138,A 93.3777,B 24.7709,C -1.7475,E1 24.8078,E2 352.7813} C_DIS
LIN {X -18.8596,Y 121.753,Z 138,A 95.0706,B 24.7712,C -1.7425,E1 24.8031,E2 351.0988} C_DIS
LIN {X -22.8793,Y 121.0622,Z 138,A 97.3932,B 24.77,C -1.7607,E1 24.7966,E2 348.7302} C_DIS
LIN {X -26.7283,Y 120.2729,Z 138,A 98.7567,B 24.7715,C -1.7376,E1 24.793,E2 347.4203} C_DIS
LIN {X -30.1546,Y 119.4578,Z 138,A 100.3107,B 24.7719,C -1.7322,E1 24.7889,E2 345.877} C_DIS
LIN {X -33.1822,Y 118.6523,Z 138,A 101.7906,B 24.7719,C -1.7318,E1 24.7849,E2 344.3959} C_DIS
LIN {X -36.2226,Y 117.7598,Z 138,A 103.3999,B 24.7716,C -1.7363,E1 24.7805,E2 342.773} C_DIS
LIN {X -40.0481,Y 116.5147,Z 138,A 105.4325,B 24.7713,C -1.7414,E1 24.7751,E2 340.7244} C_DIS
LIN {X -44.448,Y 114.9079,Z 138,A 107.3766,B 24.7722,C -1.7278,E1 24.7701,E2 338.8086} C_DIS
LIN {X -47.211,Y 113.8007,Z 138,A 108.8022,B 24.7722,C -1.7278,E1 24.7664,E2 337.3801} C_DIS
LIN {X -50.3487,Y 112.4473,Z 138,A 110.2609,B 24.7727,C -1.7195,E1 24.7627,E2 335.9377} C_DIS
LIN {X -53.4316,Y 111.0161,Z 138,A 112.0165,B 24.7724,C -1.7249,E1 24.7582,E2 334.1646} C_DIS
LIN {X -56.8563,Y 109.3022,Z 138,A 113.8079,B 24.7725,C -1.7224,E1 24.7538,E2 332.3743} C_DIS
LIN {X -60.1976,Y 107.4994,Z 138,A 115.6528,B 24.7725,C -1.7228,E1 24.7493,E2 330.523} C_DIS
LIN {X -65.039,Y 104.6412,Z 138,A 118.2514,B 24.7729,C -1.7173,E1 24.7431,E2 327.9297} C_DIS
LIN {X -68.7044,Y 102.2726,Z 138,A 120.3271,B 24.7729,C -1.7153,E1 24.7382,E2 325.8517} C_DIS
LIN {X -72.2714,Y 99.7832,Z 138,A 122.1936,B 24.7737,C -1.7042,E1 24.734,E2 324.0054} C_DIS
LIN {X -75.1873,Y 97.6056,Z 138,A 124.0768,B 24.7734,C -1.7091,E1 24.7298,E2 322.1036} C_DIS
LIN {X -78.795,Y 94.7168,Z 138,A 126.2033,B 24.7738,C -1.7033,E1 24.7252,E2 319.9829} C_DIS
LIN {X -81.9607,Y 91.9912,Z 138,A 128.1776,B 24.774,C -1.7002,E1 24.721,E2 318.0081} C_DIS
LIN {X -85.3238,Y 88.8806,Z 138,A 130.2882,B 24.7743,C -1.6943,E1 24.7168,E2 315.903} C_DIS
LIN {X -88.3236,Y 85.9003,Z 138,A 132.2866,B 24.7746,C -1.6908,E1 24.7128,E2 313.9043} C_DIS
LIN {X -91.4498,Y 82.5644,Z 138,A 134.3733,B 24.775,C -1.6837,E1 24.7089,E2 311.8255} C_DIS
LIN {X -94.1462,Y 79.4763,Z 138,A 136.3512,B 24.7751,C -1.6819,E1 24.7053,E2 309.8429} C_DIS
LIN {X -96.8932,Y 76.1022,Z 138,A 138.2799,B 24.7757,C -1.6723,E1 24.702,E2 307.9281} C_DIS
LIN {X -99.1609,Y 73.1233,Z 138,A 140.1048,B 24.7758,C -1.6712,E1 24.6989,E2 306.0969} C_DIS
LIN {X -101.6479,Y 69.6244,Z 138,A 141.976,B 24.7765,C -1.6601,E1 24.6959,E2 304.243} C_DIS
LIN {X -103.8046,Y 66.3661,Z 138,A 143.7895,B 24.7768,C -1.6548,E1 24.6932,E2 302.4332} C_DIS
LIN {X -105.688,Y 63.3239,Z 138,A 146.2399,B 24.775,C -1.6847,E1 24.6895,E2 299.8983} C_DIS
LIN {X -108.2114,Y 58.9081,Z 138,A 148.0614,B 24.7769,C -1.6536,E1 24.6872,E2 298.1416} C_DIS
LIN {X -110.2531,Y 54.9902,Z 138,A 150.0702,B 24.7774,C -1.6454,E1 24.6846,E2 296.1416} C_DIS
LIN {X -111.9777,Y 51.3859,Z 138,A 152.0308,B 24.7775,C -1.6443,E1 24.6823,E2 294.1731} C_DIS
Enddeposition()
END
